1900:
		tonUpperTimeOutFive.IN :=TRUE;
		_fbDiameterMovement.Execute :=TRUE	;	
		IF _fbDiameterMovement.PickDone THEN
			tonUpperTimeOutFive.IN :=FALSE;
			FeedBack.SecondBoxCameraDiameter:=TRUE;
			uiExecutingStep :=2000;
		END_IF
		IF tonUpperTimeOutFive.Q THEN
			_Abort :=TRUE;
			strStatus :='C# DiameterMovement Pickdone timeout';
		END_IF
2000:	//check Second Box CamaraDone
		tonUpperTimeOutFive.IN :=TRUE;
		IF info.SecondBoxCameraDiameterDone THEN
			tonUpperTimeOutFive.IN :=FALSE;
			FeedBack.SecondBoxCameraDiameter:=FALSE;
			_fbDiameterMovement.bContinue:=TRUE;
			uiExecutingStep :=2100;
		END_IF
		IF tonUpperTimeOutFive.Q THEN
			_Abort :=TRUE;
			strStatus :='C# SecondBoxCameraDiameterDone timeout';
		END_IF		
2100:	
		tonUpperTimeOutFive.IN :=TRUE;
		IF _fbDiameterMovement.Done THEN
			tonUpperTimeOutFive.IN :=FALSE;
			_fbDiameterMovement.Execute:=FALSE;
			uiExecutingStep :=2150;
		END_IF
		IF tonUpperTimeOutFive.Q THEN
			_Abort :=TRUE;
			strStatus :='_fbDiameterMovement Done timeout';
		END_IF
2150:
		IF  Input.bUpCV_BoxArrived_Sensor  AND 
			NOT Input.bUpCV_Block1Detect_Sensor  THEN
			uiExecutingStep :=2200;
		END_IF
2200:	// release box 2 from diameter camera pos
		tonUpperTimeOut.IN :=TRUE;
		tonUpperConveyorDelay.PT:=T#100MS;
		tonUpperConveyorDelay.IN := NOT Input.bUpCV_Block1Detect_Sensor ;
		IF tonUpperConveyorDelay.Q THEN	
			tonUpperConveyorDelay.IN := FALSE;
			Cylinder.List.fbUpCV_Block1.M_Extend();
			Cylinder.List.fbUpCV_DiameterPress.M_Retract();		
			Cylinder.List.fbUpCV_Block2.M_Retract();
			uiExecutingStep :=2300;
		END_IF
		IF tonUpperTimeOut.Q THEN
			_Error :=TRUE;
			strStatus := 'There is a box on Input.bUpCV_Block1Detect_Sensor '; 
		END_IF
		
		
2300:
		tonUpperTimeOut.IN :=TRUE;
		IF 	Cylinder.List.fbUpCV_DiameterPress.InRearPosition AND
			Cylinder.List.fbUpCV_Block1.InFrontPosition AND
			Cylinder.List.fbUpCV_Block2.InRearPosition THEN
			tonUpperTimeOut.IN :=FALSE;
			uiExecutingStep :=2500;
		END_IF	
		IF tonUpperTimeOut.Q THEN
			_Error :=TRUE;
			strStatus :='BlockBox1 MoveForward or BlockBox2 MoveBackward or DiameterMeasurementPressBox MoveBackward timeout';
		END_IF
2400:	//Check Box1 in FeedInBox1Detecting and Box2 leave BlockBox2Detecting
		
		tonUpperConveyorDelay.PT:=T#200MS;
		tonUpperConveyorDelay.IN := Input.bUpCV_BoxArrived_Sensor ;
		
		IF  tonUpperConveyorDelay.Q AND NOT Input.bUpCV_Block1Detect_Sensor  THEN
			tonUpperConveyorDelay.IN:=FALSE;
			Cylinder.List.fbUpCV_CamaraPress1.M_Retract();
			Cylinder.List.fbUpCV_Block3.M_Retract();
			Cylinder.List.fbUpCV_Block1.M_Extend();
			uiExecutingStep :=2500;
		END_IF
		
2500:	// Check Box1 in FeedInBox1Sensor and Box2 in BlockBox1Sensor
		tonUpperTimeOutFive.IN :=TRUE;
		tonUpperConveyorDelay.PT:=T#1000MS;
		tonUpperConveyorDelay.IN := Input.bUpCV_BoxArrived_Sensor  AND 
		(Input.bUpCV_Block1Detect_Sensor  OR NOT SecondBox);
		
		IF tonUpperConveyorDelay.Q THEN
			tonUpperTimeOutFive.IN :=FALSE;
			tonUpperConveyorDelay.IN :=FALSE;
			Cylinder.List.fbUpCV_FeedInPress1.M_Extend();
			IF SecondBox THEN
				Cylinder.List.fbUpCV_FeedInPress2.M_Extend();
			END_IF
			uiExecutingStep :=2600;
		END_IF
		IF tonUpperTimeOutFive.Q THEN
			_Error :=TRUE;
			strStatus :='FeedInBox1Detecting not have a box';
		END_IF
2600:
		tonUpperConveyorDelay.PT:=T#500MS;
		tonUpperTimeOut.IN := TRUE;
		tonUpperConveyorDelay.IN :=  Cylinder.List.fbUpCV_FeedInPress1.InFrontPosition AND
		 (Cylinder.List.fbUpCV_FeedInPress2.InFrontPosition OR NOT SecondBox);		
//		IF tonUpperConveyorDelay.IN THEN
//			iMoveConveyor:=0;
//			//Motor.list.UpCV.M_StopMotor();
//		END_IF
		IF tonUpperConveyorDelay.Q THEN
			iMoveConveyor:=0;
			tonUpperTimeOut.IN :=FALSE;
			tonUpperConveyorDelay.IN :=FALSE;
			 Cylinder.List.fbUpCV_FeedInPress1.M_Retract();
			IF SecondBox THEN
				Cylinder.List.fbUpCV_FeedInPress2.M_Retract();
			END_IF
			uiExecutingStep :=2700;
		END_IF	
		IF tonUpperTimeOut.Q THEN
			_Error :=TRUE;
			strStatus :=' Cylinder.List.fbUpCV_FeedInPress1 or Cylinder.List.fbUpCV_FeedInPress2 MoveForward timeout';
		END_IF
2700:
		tonUpperTimeOut.IN :=TRUE;
		IF TON_CheckHaveBox.IN THEN	// conveyor behind not have box feedback 0
			FeedBack.ActualNrOfBox:=0;
		ELSIF SecondBox THEN
			FeedBack.ActualNrOfBox:=2;
			ELSE
			FeedBack.ActualNrOfBox:=1;	
		END_IF
		//Cylinder.List.fbUpCV_Block1.M_Retract();
		//Cylinder.List.fbUpCV_CamaraPress2.M_Retract();
		IF NOT input.bUpCV_ReLoadDetect_Sensor  THEN
			FeedBack.InterventionRequest :=TRUE;
		END_IF
		IF// Cylinder.List.fbUpCV_Block1.InRearPosition AND
			 Cylinder.List.fbUpCV_FeedInPress1.InRearPosition AND
			Cylinder.List.fbUpCV_FeedInPress2.InRearPosition THEN
			//Cylinder.List.fbUpCV_CamaraPress2.InRearPosition THEN
			tonUpperTimeOut.IN :=FALSE;
			uiExecutingStep := 2800;
		END_IF	
		IF tonUpperTimeOut.Q THEN 
			_Error :=TRUE;
			strStatus :='FeedInPressBox1Cylinder or FeedInPressBox2Cylinder or ReadCodePressBox2Cylinder MoveBackward timeout';
		END_IF
		
2800:	//TO check the camera photo speed recoeding time
	TSaveTime 		:= TON_RecordTimer.ET;
	tRecordTimer[iArrayNumber] 			:=TSaveTime;
	tRecordFirstTimer[iArrayNumber] 	:=TSaveFirstTime;
	tRecordSecondTimer[iArrayNumber] 	:=TSaveSecondTime;
	uiExecutingStep := 2900;
2900:
	iArrayNumber := iArrayNumber+1;
	TON_RecordTimer.IN := FALSE;
	IF iArrayNumber >= 101 THEN
		bResetRecordInfo 	:=TRUE;
		iArrayNumber 		:=1;
	END_IF
	uiExecutingStep := 9999;
9999:
	bResetRecordInfo :=FALSE;
	TON_CheckHaveBox.IN :=FALSE;
	_Executed := TRUE;
				
END_CASE
	
	
IF NOT Execute THEN
	eState:=STATE_RESETTING;
END_IF
IF _Error THEN
	//FUN_UniqueErrorCodeGenerator(iErrorID := ErrorID,UinqueErrorCode=>_UniqueErrorCode);
	eState:=STATE_ERROR;
END_IF
IF _Abort OR Abort THEN
	//FUN_UniqueErrorCodeGenerator(iErrorID := ErrorID,UinqueErrorCode=>_UniqueErrorCode);
	eSTATE:=STATE_ABORTING;
END_IF
IF _Executed THEN
	eSTATE:=STATE_Done;
END_IF
END_METHOD

METHOD  M_STATE_RESETTING
VAR_INPUT
END_VAR
Error :=_Error;
Done :=_Executed;

tonUpperTimeOut.IN:=TRUE;
Motor.List.UpCV.M_MotorStop();

IF tonUpperTimeOut.Q OR NOT _Error THEN
	CASE uiResettingStep OF
		0: 
			IF _Error THEN
				Cylinder.List.fbUpCV_Block1.M_Retract();
			END_IF
			Cylinder.List.fbUpCV_FeedInPress1 .M_Retract();	
			Cylinder.List.fbUpCV_FeedInPress2.M_Retract();
			Cylinder.List.fbUpCV_DiameterPress.M_Retract();
			Cylinder.List.fbUpCV_CamaraPress1.M_Retract();	
			//UpperReadCodePressBox2Cylinder.M_Retract();	
			Cylinder.List.fbUpCV_Block2.M_Retract();	
			Cylinder.List.fbUpCV_Block3.M_Retract();	
			Cylinder.List.fbUpCV_CamaraPress4.M_Retract();
			OutPut.bCamara_Blow :=FALSE;
			_fbDiameterMovement.Execute := FALSE;
			_fbDiameterMovement.bContinue:=FALSE;
			FeedBack.InterventionRequest :=FALSE;
			FeedBack.FirstBoxCamera :=FALSE;
			FeedBack.FirstBoxCameraDiameter :=FALSE;
			FeedBack.SecondBoxCamera :=FALSE;
			FeedBack.SecondBoxCameraDiameter :=FALSE;

		
			uiResettingStep:=9999;
		
		9999:
			_ResetCompleted:=TRUE;
	END_CASE
END_IF
IF _ResetCompleted THEN
	eSTATE:=STATE_DORMANT;
END_IF
END_METHOD

END_FUNCTION_BLOCK

// ---- Library/20_MachineUnits/21_StorageArea/Service/FB_AddBoxes_v2.TcPOU
FUNCTION_BLOCK FB_AddBoxes_v2 EXTENDS FB_ObjectBase_V2
VAR_INPUT
//	UpperBoxRefillDetection		:REFERENCE TO FB_Sensor;
//	RackPusherCylinder			:REFERENCE TO FB_Cylinder;
//	RackMotor					:REFERENCE TO FB_RackMotor_V2;
//	bUpperLayerFeedInConveyor	:REFERENCE TO FB_Motor;
	Cylinder 	: REFERENCE TO UNI_CylinderList;
	Motor	 	: REFERENCE TO UNI_MotorList;
	Input 	 	: REFERENCE TO ST_InputTable;
	OutPut	 	: REFERENCE TO ST_OutputTable;
	CurrentData      : ST_SetupPara;

	ERackState	:E_RackState;
	bClearInterventionRequest : BOOL;
	_bForceUpperCV_Use		:BOOL;
END_VAR
VAR_OUTPUT
	InterventionRequest	 : BOOL;
	FeedingBoxes		:BOOL;
END_VAR
VAR
	RackMotorStationTable   : ARRAY[0..9] OF st_StationPositions;
	uiMaxRackStation :INT :=10;
//	eState :E_MethodStatus_Basic;
//	uiExecutingStep : UDINT; // This var is used to been controll STATE_EXECUTING process.
//	uiResettingStep : UDINT;
//	uiAbortingStep : UDINT;
//	_Executed :BOOL; // Executing process completed.
//	_Error : BOOL; // FB has an error.
//	_ResetCompleted : BOOL; // FB resetting completed.
//	_AbortCompleted : BOOL; // FB aborting completed.	

	tonAddBoxTimeOut	:TON;
	tonDetectSensor		:TON;
	tonConveyorTimeOut	:TON;
	tonFeedInUseAddBoxesDelay :TON;
	strStatus	:STRING;
	_Abort		:BOOL;
	uiResumeStep : UINT;
	CurrStation : UINT;
	bInterventionRequest	 : BOOL;
	trigClearInterventionRequest : R_TRIG;
	_bClearInterventionRequestLast :BOOL;
	ftrigRackStateLeaveFeedBox		:F_Trig;	
	_UniqueErrorCode : STRING;
END_VAR

A00_BasicUnits();
SUPER^.A10_StateControl();

ACTION A00_BasicUnits:
tonAddBoxTimeOut(PT:=T#120S);
tonDetectSensor(PT:=T#1S);
tonConveyorTimeOut(PT:=T#5S);
tonFeedInUseAddBoxesDelay(PT:=T#1S);
ErrorID := 2700;

InterventionRequest:=bInterventionRequest;
ftrigRackStateLeaveFeedBox(CLK := (eRackState = E_RackState.FeedBox));
IF ftrigRackStateLeaveFeedBox.Q THEN
	bInterventionRequest:=FALSE;
END_IF

FeedingBoxes := eRackState=E_RackState.FeedBox;
END_ACTION

METHOD PRIVATE M_CheckCommand : BOOL
VAR_INPUT
END_VAR
M_CheckCommand	:= true;
END_METHOD

METHOD PRIVATE M_GetCurrentStation : BOOL
VAR
	i : UINT;
	SetPos	 :LREAL;
END_VAR

VAR_OUTPUT
	uiCurrentStation	:UINT;
END_VAR
//SetPos := THIS^.fbMotor.NcToPlc.SetPos;
SetPos := arAxisCtrl_gb[AxisNo.RackMotor].Admin.Axis.NcToPlc.SetPos;
M_RefreshStationPos();
//IF  THIS^.fbMotor.Status.Homed THEN
IF arAxisCtrl_gb[AxisNo.RackMotor].Admin.Axis.Status.Homed THEN
	FOR i:=0 TO 9 BY 1 DO 
		IF SetPos> RackMotorStationTable[i].Position-5 AND SetPos< RackMotorStationTable[i].Position+5 THEN // Range should be confirm
			uiCurrentStation :=i;
			M_GetCurrentStation :=TRUE;
			RETURN;
		END_IF
	END_FOR
	
	uiCurrentStation:=99;
	M_GetCurrentStation :=FALSE;
ELSE
	M_GetCurrentStation :=FALSE;
	uiCurrentStation:=99;
END_IF
END_METHOD

METHOD PRIVATE M_MoveToStation : BOOL
VAR_INPUT
	uiStation : UINT;
END_VAR
VAR
	bDone	:BOOL;
	uiTargetPosition	:LREAL ;
END_VAR
M_RefreshStationPos();
IF uiStation>=0 AND uiStation <10 THEN
	uiTargetPosition :=RackMotorStationTable[uiStation].Position;
	
	arAxisCtrl_gb[AxisNo.RackMotor].PosMode.Acc := CurrentData.Axes.RackMotor.HalfAuto.Acceleration;
	arAxisCtrl_gb[AxisNo.RackMotor].PosMode.Dec := CurrentData.Axes.RackMotor.HalfAuto.Deceleration;
	arAxisCtrl_gb[AxisNo.RackMotor].PosMode.Jerk := CurrentData.Axes.RackMotor.HalfAuto.Jerk;
	arAxisCtrl_gb[AxisNo.RackMotor].PosMode.Velocity := CurrentData.Axes.RackMotor.HalfAuto.Velocity;
	arAxisCtrl_gb[AxisNo.RackMotor].PosMode.Position := uiTargetPosition;
	
//	THIS^.fbMotor.MoveAbs(lrPosition	:=uiTargetPosition,
//						lrVelocity 		:=GVL.MotorCore[AxisNo.RackMotor].VCC,
//						lrAcceleration	:=GVL.MotorCore[AxisNo.RackMotor].ACC,
//						lrDeceleration	:=GVL.MotorCore[AxisNo.RackMotor].DCC,
//						lrJerk			:=GVL.MotorCore[AxisNo.RackMotor].Jerk,
//						BufferMode		:=MC_BufferMode.MC_Aborting);
	//THIS^.fbMotor.GetCmdDoneStatus(bMotionCmdDone=>bDone);
ELSE
	M_MoveToStation :=FALSE;
	RETURN;
END_IF
END_METHOD

METHOD PRIVATE M_RefreshStationPos : BOOL
VAR_INPUT
END_VAR
VAR
	i: UINT;
	position : ST_PositionTable;
END_VAR
FOR i := 0 TO 9 DO
	position :=FUN_GetPositionTableData(PositionName:='W',Index:=i,Clip:=0);
RackMotorStationTable[i].Position:= position.X_Pos;
END_FOR
	M_RefreshStationPos :=TRUE;

// todo : update position of each stations
//FOR i:=1 TO 200 BY 1 DO
//	FOR iIndex:=0 TO 9 BY 1 DO
//		IF 		
//			DAS_CoreSys.MachineControl.CurrentData.PositionTable[i].Index= iIndex AND
//			DAS_CoreSys.MachineControl.CurrentData.PositionTable[i].Zone ='W' THEN
//			RackMotorStationTable[iIndex].Position := DAS_CoreSys.MachineControl.CurrentData.PositionTable[i].X_Pos;

//			StationsPosition[iIndex]:=RackMotorStationTable[i].Position;
//		ELSE
//			M_RefreshStationPos :=FALSE;
//		END_IF
//	END_FOR
//END_FOR
END_METHOD

METHOD  M_STATE_ABORTED
VAR_INPUT
END_VAR
Error :=TRUE;
Busy :=FALSE;
Done := FALSE;
Status :=strStatus;
UniqueErrorCode:=_UniqueErrorCode;
if not Execute then
	eState := STATE_RESETTING;
END_IF
IF Execute AND Reset THEN
	_Abort := FALSE;
	uiExecutingStep:=uiResumeStep;
	eState:=STATE_EXECUTING;
END_IF
END_METHOD

METHOD  M_STATE_ABORTING
VAR_INPUT
END_VAR
CASE uiAbortingStep of
 0:
 	Cylinder.List.fbStackPush.M_Reset();

	//RackMotor.fbMotor.Reset();	
	
	uiAbortingStep:=9999;
	
9999:	
	_AbortCompleted:=TRUE;
END_CASE

IF	 _AbortCompleted THEN
	eSTATE:=STATE_ABORTED;
END_IF
END_METHOD

METHOD  M_STATE_DONE
VAR_INPUT
END_VAR
Busy := FALSE;
Done := TRUE;
IF NOT Execute THEN
	eState := STATE_RESETTING;
END_IF
END_METHOD

METHOD  M_STATE_DORMANT
VAR_INPUT
END_VAR
VAR
END_VAR
Busy    := FALSE;
Done    := FALSE;
Aborted := FALSE;
Error   := FALSE;
strStatus  := 'No error';
uiExecutingStep := 0;
uiResettingStep := 0;
uiAbortingStep:=0;
uiResumeStep:=0;
_ResetCompleted := FALSE;
_Abort := _Executed := _Error:= _ResetCompleted:=_AbortCompleted:=FALSE;
tonAddBoxTimeOut.IN :=FALSE;
tonDetectSensor.IN:=FALSE;
tonFeedInUseAddBoxesDelay.IN :=FALSE;
_UniqueErrorCode :='0';

IF Execute  THEN 
	IF eRackState = E_RackState.FeedBox THEN
		eState:= STATE_ERROR;
		strStatus :='Rack occupied by user Push FeedButton';
		
	ELSIF  Input.bUpCV_ReLoadDetect_Sensor THEN
		_Executed :=TRUE;
		eState	:= STATE_Done;
	ELSE
		eState := STATE_EXECUTING;
	END_IF	
END_IF
END_METHOD

METHOD  M_STATE_ERROR
VAR_INPUT
END_VAR
Error := TRUE;
Busy :=FALSE;
Status :=strStatus;
UniqueErrorCode:=_UniqueErrorCode;
IF NOT Execute THEN
	eSTATE :=STATE_RESETTING;
END_IF
END_METHOD

METHOD  M_STATE_EXECUTING
VAR_INPUT
END_VAR
VAR_INST
	uiTargetStation	: UINT;
	bMoveConveyor	:BOOL;
END_VAR
VAR
	bMotionDone : BOOL;
	
END_VAR
Busy := TRUE; 
IF NOT _bForceUpperCV_Use THEN
	IF bMoveConveyor THEN
		Motor.List.UpCV.M_MoveForward();	
//	ELSE		
//		Motor.List.UpCV.M_MotorStop();	
	END_IF
END_IF
CASE uiExecutingStep OF			
	0:		//check command
		tonAddBoxTimeOut.IN:=FALSE;
		tonFeedInUseAddBoxesDelay.IN :=TRUE;
			IF M_CheckCommand() THEN
				IF tonFeedInUseAddBoxesDelay.Q THEN
					tonFeedInUseAddBoxesDelay.IN :=FALSE;
					uiExecutingStep	:= 10 ;
				END_IF
			ELSE
				strStatus := 'Wrong command, check the command setting';
				_Error := TRUE;
			END_IF
	10:

		IF 	NOT	Motor.List.UpCV.InBackWard THEN
			uiExecutingStep	:= 100 ;
		END_IF
		//todo : Add timeout
		
 	100:	//release cylinder, check rackmotor currentStation
		tonAddBoxTimeOut.IN:=TRUE;
		tonDetectSensor.IN:=FALSE;
		Cylinder.List.fbStackPush.M_Retract();
		M_GetCurrentStation(uiCurrentStation =>CurrStation);
		
		IF	Cylinder.List.fbStackPush.InRearPosition THEN
		 CASE CurrStation OF
			0 ,99 :
				uiTargetStation:=1;				
			1,2,3,4,5,6,7,8,9 :
				uiTargetStation :=CurrStation;	
			
			ELSE // Error
	
	 	 END_CASE
		END_IF
		
		uiExecutingStep	:= 200 ;
		IF tonAddBoxTimeOut.Q THEN
			strStatus := 'RackPusher move back timeout';
			uiResumeStep:=100;
            _Abort := TRUE;
		END_IF
		
	200:	//check rackmotor station 
		tonDetectSensor.IN :=FALSE;
		IF uiTargetStation<10 THEN
			M_MoveToStation(uiTargetStation);
			uiExecutingStep := 210;	
		ELSE
			uiExecutingStep := 500;	
		END_IF
		
	
	210:
		tonAddBoxTimeOut.IN:=TRUE;
		bMotionDone:= arAxisStatus_gb[AxisNo.RackMotor].Admin._OpModeAck = ModePosAbs AND arAxisStatus_gb[AxisNo.RackMotor].Admin.CmdDone;
	//	RackMotor.fbMotor.GetCmdDoneStatus(bMotionCmdDone=>bMotionDone);
		M_GetCurrentStation(uiCurrentStation =>CurrStation);
	//CurrStation:= RackMotor.P_CurrentStattion;
		IF bMotionDone AND uiTargetStation = CurrStation THEN
			tonAddBoxTimeOut.IN:=FALSE;
			uiExecutingStep := 300;	
		END_IF
		IF tonAddBoxTimeOut.Q THEN
			strStatus := 'Rackmotor moving timeout';
            _Error := TRUE;
		END_IF
		
	300:	//Cylinder moveforward
		tonAddBoxTimeOut.IN:=TRUE;
		Cylinder.List.fbStackPush.M_Extend();
		//bUpperLayerFeedInConveyor.M_ForwardMotor('');
		bMoveConveyor :=TRUE; //Move conveyor motor forward
		IF  Motor.List.UpCV.InForWard THEN	// make sure upperCV release force use
			IF Cylinder.List.fbStackPush.InFrontPosition THEN
				tonAddBoxTimeOut.IN:=FALSE;
				uiExecutingStep := 400;
			END_IF
		END_IF
		IF tonAddBoxTimeOut.Q THEN
			strStatus := 'RackPusher move forward timeout';
			uiResumeStep:=300;
            _Abort := TRUE;
		END_IF
		
	400:	//check refillsensor have refill
		tonDetectSensor.IN:= NOT Input.bUpCV_ReLoadDetect_Sensor;
		Cylinder.List.fbStackPush.M_Retract();
		IF Cylinder.List.fbStackPush.InRearPosition THEN
			IF Input.bUpCV_ReLoadDetect_Sensor THEN
				uiExecutingStep :=500;
			ELSIF tonDetectSensor.Q THEN
				uiTargetStation := CurrStation+1;		
				uiExecutingStep :=200;
			END_IF
		END_IF
		
	500:	//確認氣缸是否在後，Done
		tonAddBoxTimeOut.IN:=TRUE;
			//bUpperLayerFeedInConveyor.M_StopMotor(''); 
			//bMoveConveyor :=FALSE;// Stop Conveyor
			tonAddBoxTimeOut.IN:=FALSE;
			IF uiTargetStation>=9 THEN
				uiExecutingStep :=600;
			ELSE
				bMoveConveyor :=FALSE;
				Motor.List.UpCV.M_MotorStop();	
				uiExecutingStep :=1000;
			END_IF
		
		
		IF tonAddBoxTimeOut.Q THEN
			strStatus := 'RackPusher move back timeout';
			uiResumeStep:=400;
            _Abort := TRUE;
		END_IF
	600:
		tonAddBoxTimeOut.IN:=FALSE	;
		 M_MoveToStation(0);
		 uiExecutingStep:=610;
		 
	610:	
		M_GetCurrentStation(uiCurrentStation =>CurrStation);
		tonAddBoxTimeOut.IN:=TRUE;
		bMotionDone:=arAxisStatus_gb[AxisNo.RackMotor].Admin._OpModeAck = ModePosAbs AND arAxisStatus_gb[AxisNo.RackMotor].Admin.CmdDone;
		IF bMotionDone AND 0 = CurrStation THEN
			bInterventionRequest	 :=TRUE;
			tonAddBoxTimeOut.IN:=FALSE	;
			bMoveConveyor :=FALSE;
			Motor.List.UpCV.M_MotorStop();	
			uiExecutingStep:=1000;
		END_IF
 		IF tonAddBoxTimeOut.Q THEN
			strStatus := 'RackPusher move back timeout';
			uiResumeStep:=400;
            _Abort := TRUE;
		END_IF
	1000:
		bMoveConveyor :=FALSE;// Stop Conveyor
		uiExecutingStep:=1100;
		
	1100:		
		_Executed := TRUE;
	
		
//		strStatus := 'Rack is empty';
//		_Error :=TRUE;
	
	
END_CASE

IF NOT Execute THEN
	eSTATE :=STATE_RESETTING;
END_IF
IF _Executed THEN
	eSTATE := STATE_DONE;
END_IF
IF _Error THEN
	//FUN_UniqueErrorCodeGenerator(iErrorID := ErrorID,UinqueErrorCode=>_UniqueErrorCode);
	eSTATE:=STATE_ERROR;
END_IF
IF _Abort OR Abort THEN
	//FUN_UniqueErrorCodeGenerator(iErrorID := ErrorID,UinqueErrorCode=>_UniqueErrorCode);
	eSTATE:=STATE_ABORTING;
END_IF
END_METHOD

METHOD  M_STATE_RESETTING
VAR_INPUT
END_VAR

VAR
	bMotionDone : BOOL;
END_VAR
CASE uiResettingStep OF
	0:
		tonAddBoxTimeOut.IN:=FALSE;		
		tonDetectSensor.IN:=FALSE;
		Cylinder.List.fbStackPush.M_Retract();

		IF Cylinder.List.fbStackPush.InRearPosition THEN
		uiResettingStep :=100;
		END_IF
		
	100:
		arAxisCtrl_gb[AxisNo.RackMotor].Admin._OpMode.en := E_AXIS_MODE.ModeAH;
		//RackMotor.fbMotor.Stop(0,0);
		//RackMotor.fbMotor.GetCmdDoneStatus(bMotionCmdDone=>bMotionDone);
		Motor.List.UpCV.M_MotorStop();
		uiResettingStep := 200;

		
	200:
		 Error :=false;
		_ResetCompleted := TRUE;
END_CASE

IF _ResetCompleted THEN
	eState := STATE_DORMANT;
END_IF
END_METHOD

END_FUNCTION_BLOCK

// ---- Library/20_MachineUnits/21_StorageArea/Service/FB_BoxSupplyCtrl.TcPOU
FUNCTION_BLOCK FB_BoxSupplyCtrl EXTENDS FB_ObjectBase_V2
VAR_INPUT
//    Execute    :BOOL;   // True : This prog will start.
//    Abort      :BOOL;   // True : This prog will be abort.
//    Reset      :BOOL;   // True : This prog will be reset.
//    ObjectName :STRING; // Set this fb name(About it's action)

//	SupplyBTN 				:REFERENCE TO FB_Button;			//2nd machine
//	RackMotor				:REFERENCE TO FB_RackMotor_V2;
//	BoxesPusherCylinder		:REFERENCE TO FB_Cylinder;


	Cylinder				:REFERENCE TO UNI_CylinderList;
	Input 					:REFERENCE TO ST_InputTable;
	Output					:REFERENCE TO ST_OutputTable;
	StroageRegionMode 		:E_UnitMode;
	bAddsBoxRequest 		: BOOL;
	AddBoxes_Status			:ST_AutoAddsBoxesStatus;
	AddBoxes_Ctrl			:ST_AutoAddsBoxesCommand;
	CurrentData 			: ST_SetupPara;
	
END_VAR

VAR_OUTPUT
	RackState : E_RackState;
	AxisRackMotorBTNHomeRequest	:BOOL;
//    Busy    :BOOL;        // True : This prog is running.
//    Done    :BOOL;        // True : Command has been executed.
//    Aborted :BOOL;        // True : This prog is aborted.
//    Error   :BOOL;        // True : This prog has an error.
//    ErrorID :UINT;       // Output ErrorID
//    Status  :T_MaxString; // Output this prog status by string(255bytes)
END_VAR

VAR
//    eState :E_MethodStatus_Basic;
//	uiExecutingStep : UDINT; // This var is used to been controll STATE_EXECUTING process.
//	uiResettingStep : UDINT;
//	uiAbortingStep : UDINT;
//	_Executed :BOOL; // Executing process completed.
//	_Error : BOOL; // FB has an error.
//	_ResetCompleted : BOOL; // FB resetting completed.
//	_AbortCompleted : BOOL; // FB aborting completed.
	RackMotorStationTable   : ARRAY[0..9] OF st_StationPositions;
	uiMaxRackStation :INT :=10;
	_Abort		: BOOL;
	strStatus	: STRING;
	uiResumeStep : UINT;
	ExcutingStep :E_RackState;
	trigBTN			:R_TRIG;
	trigRequest		:R_TRIG;
	tonBtnCtrl		:ton;
	tonBtnMotorCtrl	:ton;
	tonBlinkTimer :TON;
	tonBlink_Internal :TIME :=T#500MS;

END_VAR

A00_BasicUnits();
SUPER^.A10_StateControl();

ACTION A00_BasicUnits:
tonBtnCtrl(PT:=T#5S);
tonBtnMotorCtrl(PT :=T#30S);
ErrorID := 2800;
END_ACTION

METHOD GetModelState
VAR_OUTPUT
    xDone    :BOOL;
    xBusy    :BOOL;
    xError   :BOOL;
    xAborted :BOOL;
    iErrorID :UDINT;
	UniqueErrorCode : STRING;
END_VAR
xDone    := Done;
xBusy    := Busy;
xError   := Error;
xAborted := Abort;
iErrorID := ErrorID;
END_METHOD

METHOD GetName : STRING
GetName := ObjectName;
END_METHOD

METHOD PRIVATE M_Blink : BOOL
VAR_INPUT
	
END_VAR
tonBlinkTimer(IN :=NOT tonBlinkTimer.Q,
				PT := tonBlink_Internal);
IF tonBlinkTimer.Q THEN
	Output.bStorage_StackPushPbLamp := NOT Output.bStorage_StackPushPbLamp;
END_IF
END_METHOD

METHOD PRIVATE M_GetCurrentStation : BOOL
VAR
	i : UINT;
	SetPos	 :LREAL;
END_VAR

VAR_OUTPUT
	uiCurrentStation	:UINT;
END_VAR
//SetPos := THIS^.fbMotor.NcToPlc.SetPos;
SetPos := arAxisCtrl_gb[AxisNo.RackMotor].Admin.Axis.NcToPlc.SetPos;
M_RefreshStationPos();
//IF  THIS^.fbMotor.Status.Homed THEN
IF arAxisCtrl_gb[AxisNo.RackMotor].Admin.Axis.Status.Homed THEN
	FOR i:=0 TO 9 BY 1 DO 
		IF SetPos> RackMotorStationTable[i].Position-5 AND SetPos< RackMotorStationTable[i].Position+5 THEN // Range should be confirm
			uiCurrentStation :=i;
			M_GetCurrentStation :=TRUE;
			RETURN;
		END_IF
	END_FOR
	
	uiCurrentStation:=99;
	M_GetCurrentStation :=FALSE;
ELSE
	M_GetCurrentStation :=FALSE;
	uiCurrentStation:=99;
END_IF
END_METHOD

METHOD PRIVATE M_MoveToStation : BOOL
VAR_INPUT
	uiStation : UINT;
END_VAR
VAR
	bDone	:BOOL;
	uiTargetPosition	:LREAL ;
END_VAR
M_RefreshStationPos();
IF uiStation>=0 AND uiStation <10 THEN
	uiTargetPosition :=RackMotorStationTable[uiStation].Position;
	
	arAxisCtrl_gb[AxisNo.RackMotor].PosMode.Acc := CurrentData.Axes.RackMotor.HalfAuto.Acceleration;
	arAxisCtrl_gb[AxisNo.RackMotor].PosMode.Dec := CurrentData.Axes.RackMotor.HalfAuto.Deceleration;
	arAxisCtrl_gb[AxisNo.RackMotor].PosMode.Jerk := CurrentData.Axes.RackMotor.HalfAuto.Jerk;
	arAxisCtrl_gb[AxisNo.RackMotor].PosMode.Velocity := CurrentData.Axes.RackMotor.HalfAuto.Velocity;
	arAxisCtrl_gb[AxisNo.RackMotor].PosMode.Position := uiTargetPosition;
	
//	THIS^.fbMotor.MoveAbs(lrPosition	:=uiTargetPosition,
//						lrVelocity 		:=GVL.MotorCore[AxisNo.RackMotor].VCC,
//						lrAcceleration	:=GVL.MotorCore[AxisNo.RackMotor].ACC,
//						lrDeceleration	:=GVL.MotorCore[AxisNo.RackMotor].DCC,
//						lrJerk			:=GVL.MotorCore[AxisNo.RackMotor].Jerk,
//						BufferMode		:=MC_BufferMode.MC_Aborting);
	//THIS^.fbMotor.GetCmdDoneStatus(bMotionCmdDone=>bDone);
ELSE
	M_MoveToStation :=FALSE;
	RETURN;
END_IF
END_METHOD

METHOD PRIVATE M_RefreshStationPos : BOOL
VAR_INPUT
END_VAR
VAR
	i: UINT;
	position : ST_PositionTable;
END_VAR
FOR i := 0 TO 9 DO
	position :=FUN_GetPositionTableData(PositionName:='W',Index:=i,Clip:=0);
RackMotorStationTable[i].Position:= position.X_Pos;
END_FOR
	M_RefreshStationPos :=TRUE;

// todo : update position of each stations
//FOR i:=1 TO 200 BY 1 DO
//	FOR iIndex:=0 TO 9 BY 1 DO
//		IF 		
//			DAS_CoreSys.MachineControl.CurrentData.PositionTable[i].Index= iIndex AND
//			DAS_CoreSys.MachineControl.CurrentData.PositionTable[i].Zone ='W' THEN
//			RackMotorStationTable[iIndex].Position := DAS_CoreSys.MachineControl.CurrentData.PositionTable[i].X_Pos;

//			StationsPosition[iIndex]:=RackMotorStationTable[i].Position;
//		ELSE
//			M_RefreshStationPos :=FALSE;
//		END_IF
//	END_FOR
//END_FOR
END_METHOD

METHOD  M_STATE_ABORTED
VAR_INPUT
END_VAR
ERROR :=TRUE;
Busy    := FALSE;
Aborted := TRUE;
Status := strStatus;

IF NOT Execute THEN
	eSTATE:=STATE_RESETTING;
END_IF

IF Execute AND Reset THEN
	uiExecutingStep :=uiResumeStep;
	eSTATE:=STATE_EXECUTING;
END_IF
END_METHOD

METHOD  M_STATE_ABORTING
VAR_INPUT
END_VAR
CASE uiAbortingStep OF
	0 :
		uiAbortingStep:=9999;
	
	9999:	_AbortCompleted:=TRUE;
END_CASE

IF _AbortCompleted THEN	
	eSTATE :=STATE_ABORTED;
END_IF
END_METHOD

METHOD  M_STATE_DONE
VAR_INPUT
END_VAR
Busy 	:= FALSE;
Done	:=TRUE;

IF NOT Execute THEN
	eSTATE:=STATE_RESETTING;
END_IF
END_METHOD

METHOD  M_STATE_DORMANT
VAR_INPUT
END_VAR
Busy            := FALSE;
Done            := FALSE;
Aborted         := FALSE;
Error           := FALSE;
ErrorID         := 0;
Status          := '';
_ResetCompleted := FALSE;
_Error          := FALSE;
_Executed       := FALSE;
strStatus :='No Error';
uiExecutingStep :=uiResettingStep :=uiResumeStep :=0;

IF Execute THEN
	eSTATE:=STATE_EXECUTING;
END_IF
END_METHOD

METHOD  M_STATE_ERROR
VAR_INPUT
END_VAR
ERROR   :=TRUE;
Busy	:=FALSE;
Status := strStatus;
M_TurnOff();
RackState:= E_RackState.idle; // Useless so far
AxisRackMotorBTNHomeRequest :=false;
IF NOT Execute OR Reset THEN // Execute will always on , therefor Reset is only way to recovery from error	
	eSTATE:=STATE_RESETTING;
END_IF
END_METHOD

METHOD  M_STATE_EXECUTING
VAR_INPUT
END_VAR

VAR_INST
	uiTransitingStep : UINT;
	uiTargetStation :UINT :=0;
	bFreeState	  :BOOL;
END_VAR

VAR
	bMotionDone			:BOOL;
	_uiCurrentStation	:UINT;
END_VAR
Busy :=TRUE;	
//IF SupplyBTN.P_IsBTNRef THEN			//2nd machine 
//	trigBTN(CLK:= (SupplyBTN.P_ButtonState));
//END_IF //Make sure BTN is referenced otherwise exception occur

	trigBTN(CLK:= ( Input.bStorage_StackPushPb));
trigRequest(CLK :=(AddBoxes_Status.InterventionRequest AND bFreeState));

// Force state control
IF AddBoxes_Status.Busy OR AddBoxes_Status.Done  THEN	
	ExcutingStep := E_RackState.AddBoxes;
	
ELSIF StroageRegionMode = E_UnitMode.MANUAL AND
	arAxisCtrl_gb[AxisNo.RackMotor].Admin.Axis.Status.HasJob AND
//	  rackmotor.fbMotor.Status.HasJob AND 
	  NOT (ExcutingStep = E_RackState.FeedBox) THEN	
			ExcutingStep := E_RackState.ManualCtrl;

ELSIF	StroageRegionMode = E_UnitMode.MANUAL AND 
		NOT Cylinder.List.fbStackPush.InRearPosition AND
//		BoxesPusherCylinder.P_IsMoving AND 
		NOT	(ExcutingStep = E_RackState.FeedBox) THEN	
			ExcutingStep := E_RackState.ManualCtrl;

			
END_IF

RackState := ExcutingStep;

CASE ExcutingStep OF
	

	E_RackState.idle:
		;	
	E_RackState.AddBoxes:
		//Service AddBox working
		M_TurnOff();
		bFreeState:=FALSE;
		IF NOT AddBoxes_Ctrl.Execute AND NOT AddBoxes_Status.Error  THEN
        	ExcutingStep := E_RackState.Free;
    	END_IF
		
	E_RackState.ManualCtrl:
	//Stroage area in manual and Rack is moving
		M_TurnOff();
		bFreeState:=FALSE;
		IF NOT arAxisCtrl_gb[AxisNo.RackMotor].Admin.Axis.Status.HasJob AND Cylinder.List.fbStackPush.InRearPosition THEN
            ExcutingStep := E_RackState.Free;
        END_IF
		
	E_RackState.FeedBox:
	// FeedBox mode , 
		M_Blink();
		bFreeState:=FALSE;
		AxisRackMotorBTNHomeRequest :=false;
			IF	trigBTN.Q THEN				
				ExcutingStep :=E_RackState.TransitingFree;	
			END_IF
			
	E_RackState.Free:
	// Rack is free , User is allow to ask to suply box by push the suplyBTN
		M_TurnOn();
		bFreeState:=TRUE;
			 IF trigBTN.Q OR trigRequest.Q THEN
				 uiTransitingStep:=0;
				 ExcutingStep := E_RackState.TransitingFeedBox;
			 END_IF

	E_RackState.TransitingFree:
			 IF NOT AddBoxes_Status.InterventionRequest THEN
				 ExcutingStep :=E_RackState.Free;	
			 END_IF
		
	E_RackState.TransitingFeedBox:
	//Transition step , from Free to FeedBox
		//M_Blink();
		M_TurnOff();
		bFreeState:=FALSE;
		AxisRackMotorBTNHomeRequest :=TRUE;
		// todo : if transition step needs different indication of BTN behavior?
		CASE uiTransitingStep OF
		0:
			tonBtnCtrl.IN	:=FALSE;
			tonBtnMotorCtrl.IN :=FALSE;
			uiTransitingStep:=5;
			M_GetCurrentStation(uiCurrentStation =>_uiCurrentStation);
			IF uiTargetStation = _uiCurrentStation THEN
				uiTransitingStep :=30;
			END_IF
			
		5:	//Move cylinder back
			tonBtnCtrl.IN:=TRUE;			
			Cylinder.List.fbStackPush.M_Retract();
			IF Cylinder.List.fbStackPush.InRearPosition AND NOT arAxisCtrl_gb[AxisNo.RackMotor].Admin.Axis.Status.HasJob THEN 
				tonBtnCtrl.IN :=FALSE;
				uiTransitingStep :=10;
			END_IF
			IF tonBtnCtrl.Q THEN
				_Error:= TRUE;
				StrStatus :='Cylinder MoveBackward timeout';
			END_IF
		10:	// Rackmotor move to station 0
			tonBtnMotorCtrl.IN :=TRUE;
			M_MoveToStation(uiTargetStation);
			IF arAxisCtrl_gb[AxisNo.RackMotor].Admin.Axis.Status.HasJob THEN
				tonBtnMotorCtrl.IN :=FALSE;
			uiTransitingStep :=20;
			END_IF
			IF tonBtnMotorCtrl.Q THEN
				_Error :=TRUE;
				StrStatus :='RackMotor MoveToStation timeout';
			END_IF
		20:	// check currentstation 
			tonBtnMotorCtrl.IN :=TRUE;
//			bMotionDone :=rackmotor.fbMotor.Status.InTargetPosition;
			bMotionDone :=arAxisCtrl_gb[AxisNo.RackMotor].Admin.Axis.Status.InTargetPosition;
			M_GetCurrentStation(uiCurrentStation =>_uiCurrentStation);
			IF bMotionDone  AND uiTargetStation = _uiCurrentStation THEN
				
				uiTransitingStep :=30;
			END_IF
			IF tonBtnMotorCtrl.Q THEN
				_Error :=TRUE;
				StrStatus :='RackMotor currentStation timeout';
			END_IF
		30:
			tonBtnMotorCtrl.IN :=FALSE;
			ExcutingStep := E_RackState.FeedBox;
			AxisRackMotorBTNHomeRequest :=FALSE;
		END_CASE
		


END_CASE
	
IF NOT Execute THEN
	eState:=STATE_RESETTING;
END_IF
IF _Error THEN
	eState:=STATE_ERROR;
END_IF
IF _Abort THEN
	eSTATE:=STATE_ABORTING;
END_IF
IF _Executed THEN
	eSTATE:=STATE_Done;
END_IF
END_METHOD

METHOD  M_STATE_RESETTING
VAR_INPUT
END_VAR
Error :=FALSE;
Done :=FALSE;
Busy := FALSE;
AxisRackMotorBTNHomeRequest :=FALSE;
tonBtnCtrl.IN := FALSE;
tonBtnMotorCtrl.IN := FALSE;
M_TurnOff();
CASE uiResettingStep OF
	
	0:
		uiResettingStep:=9999;


	9999:
		_ResetCompleted:=TRUE;
END_CASE
IF _ResetCompleted THEN
	eSTATE:=STATE_DORMANT;
END_IF
END_METHOD

METHOD PRIVATE M_TurnOff : BOOL
VAR_INPUT
END_VAR
Output.bStorage_StackPushPbLamp := false;
END_METHOD

METHOD PRIVATE M_TurnOn : BOOL
VAR_INPUT
END_VAR
Output.bStorage_StackPushPbLamp := true;
END_METHOD

END_FUNCTION_BLOCK

// ---- Library/20_MachineUnits/23_ShippingArea/FB_ShippingArea.TcPOU
FUNCTION_BLOCK FB_ShippingArea EXTENDS FB_ModeBase_V2 IMPLEMENTS I_UnitState
VAR_INPUT
	FanucRobot : REFERENCE TO FB_FanucRobot_Basic;
	Service : REFERENCE TO ST_ShippingService;
	INPUT       : REFERENCE TO ST_InputTable;
	Motor    : REFERENCE TO UNI_MotorList;
    Reset            : REFERENCE TO BOOL;
	Stop :  REFERENCE TO BOOL;
    bStopMem :  REFERENCE TO BOOL;
END_VAR
VAR_OUTPUT
	Homed : BOOL;
	RobotResetCMD : BOOL;
END_VAR
VAR
	fbShippingRobot_TransmitCVEnd :FB_ShippingRobot_TransmitCVEnd;
	fbShippingRobot_Left : FB_ShippingRobot_Left;
	fbShippingRobot_Right : FB_ShippingRobot_Right;
	fbShippingHoming : FB_ShippingHoming;
END_VAR

SUPER^();

IF __ISVALIDREF(PackTag) THEN
    eModeCommand  := PackTag.Command.UnitMode;
    eStateCommand := PackTag.Command.CntrlCmd;
ELSE
    RETURN;
END_IF

ACTION A00_Service:
fbShippingRobot_TransmitCVEnd(
	Execute:= Service.AutoMode_ShippingRobot_TransmitCVEnd.Command.Execute, 
	Abort:= Service.AutoMode_ShippingRobot_TransmitCVEnd.Command.Abort, 
	Reset:= Reset, 
	ObjectName:= 'Shipping Fanuc Robot TransmitCVEnd', 
	INPUT:=INPUT,
	Motor :=Motor,
	Busy=> Service.AutoMode_ShippingRobot_TransmitCVEnd.Status.Busy, 
	Done=> Service.AutoMode_ShippingRobot_TransmitCVEnd.Status.Done, 
	Aborted=> , 
	Error=> Service.AutoMode_ShippingRobot_TransmitCVEnd.Status.Error, 
	ErrorID=> , 
	Status=> Service.AutoMode_ShippingRobot_TransmitCVEnd.Status.Status, 
	UniqueErrorCode=> , 
	Robot:= FanucRobot, 
	Info:= Service.AutoMode_ShippingRobot_TransmitCVEnd.Info, 
	Stop:= bStopMem);
	
fbShippingRobot_Left(
	Execute:= service.AutoMode_ShippingRobot_Left.Command.Execute, 
	Abort:= Service.AutoMode_ShippingRobot_Left.Command.Abort, 
	Reset:= Reset, 
	ObjectName:= 'Shipping Fanuc Robot Left', 
	Busy=> Service.AutoMode_ShippingRobot_Left.Status.Busy, 
	Done=> Service.AutoMode_ShippingRobot_Left.Status.Done, 
	Aborted=> , 
	Error=> Service.AutoMode_ShippingRobot_Left.Status.Error, 
	ErrorID=> , 
	Status=> Service.AutoMode_ShippingRobot_Left.Status.Status, 
	UniqueErrorCode=> , 
	Robot:= FanucRobot, 
	Info:= Service.AutoMode_ShippingRobot_Left.Info, 
	Stop:=bStopMem);
	
fbShippingRobot_Right(
	Execute:= Service.AutoMode_ShippingRobot_Right.Command.Execute, 
	Abort:= Service.AutoMode_ShippingRobot_Right.Command.Abort, 
	Reset:= Reset, 
	ObjectName:= 'Shipping Fanuc Robot Right', 
	Busy=> Service.AutoMode_ShippingRobot_Right.Status.Busy, 
	Done=> Service.AutoMode_ShippingRobot_Right.Status.Done, 
	Aborted=> , 
	Error=> Service.AutoMode_ShippingRobot_Right.Status.Error, 
	ErrorID=> , 
	Status=> Service.AutoMode_ShippingRobot_Right.Status.Status, 
	UniqueErrorCode=> , 
	Robot:= FanucRobot, 
	Info:= Service.AutoMode_ShippingRobot_Right.Info, 
	Stop:= bStopMem);
	
fbShippingHoming(
	xDone=> , 
	xBusy=> , 
	xError=> , 
	xExecute:= , 
	xAbort:= , 
	FanucRobot:= FanucRobot, 
	Homed:= Homed, 
	xAborted=> , 
	iErrorID=> , 
	ErrorMsg=> , 
	RobotResetCMD=> RobotResetCMD);
END_ACTION

METHOD M_Aborted
M_StateComplete();
END_METHOD

METHOD M_Aborting
M_StateComplete();
END_METHOD

METHOD M_Clearing
M_StateComplete();
END_METHOD

METHOD M_Complete
M_StateComplete();
END_METHOD

METHOD M_Completing
M_StateComplete();
END_METHOD

METHOD M_Execute
CASE eModeCurrent OF
	E_UnitMode.Manual:
		;
	E_UnitMode.Auto:
		;
END_CASE
A00_Service();
//M_StateComplete();
END_METHOD

METHOD M_Held
M_StateComplete();
END_METHOD

METHOD M_Holding
M_StateComplete();
END_METHOD

METHOD M_Idle
M_StateComplete();
END_METHOD

METHOD M_Resetting
M_StateComplete();
END_METHOD

METHOD M_StartHoming
VAR_INPUT
END_VAR
fbShippingHoming.xExecute := TRUE;
END_METHOD

METHOD M_Starting
M_StateComplete();
END_METHOD

METHOD M_StopHoming
VAR_INPUT
END_VAR
fbShippingHoming.xExecute := False;
END_METHOD

METHOD M_Stopped
M_StateComplete();
END_METHOD

METHOD M_Stopping
M_StateComplete();
END_METHOD

METHOD M_Suspended
M_StateComplete();
END_METHOD

METHOD M_Suspending
M_StateComplete();
END_METHOD

METHOD M_Undefined
M_StateComplete();
END_METHOD

METHOD M_Unholding
M_StateComplete();
END_METHOD

METHOD M_Unsuspending
M_StateComplete();
END_METHOD

END_FUNCTION_BLOCK

// ---- Library/20_MachineUnits/23_ShippingArea/Service/FB_ShippingRobot_TransmitCVEnd.TcPOU
FUNCTION_BLOCK FB_ShippingRobot_TransmitCVEnd EXTENDS FB_RobotRegionMove_BufferArea
VAR_INPUT
	INPUT       : REFERENCE TO ST_InputTable;
	Motor    	: REFERENCE TO UNI_MotorList;
END_VAR
VAR_OUTPUT
END_VAR
VAR
	//Area : E_RobotArea := E_RobotArea.TransmitCV_End;
	SensorToBeCheck :BIT;
	ConveyorMotor	: REFERENCE TO FB_Motor ;
	tonBoxArriveDelay 	: TON;
END_VAR

SUPER^.A10_StateControl();
A00_BasicUnits();
Area := E_RobotArea.TransmitCV_End;

ACTION A00_BasicUnits:
tonTimeOut(PT:=T#60S);
tonBoxArriveDelay(PT:=T#1S);

ErrorID:=2250;
END_ACTION

METHOD M_CheckCommand : BOOL // True : Command is useful
VAR_INPUT
END_VAR
VAR
	
END_VAR
// Check command paremeter is correct

THIS^.Get :=TRUE; // For this service , robot only pick box from conveyor
UseA := TRUE; // Only clip A avaliable
UseB := FALSE; // No clipB 	
		
	
	
CASE 	LREAL_TO_INT(Info.A_Position) OF	
	
1: // Pick box from Samesize conveyor
	SensorToBeCheck :=INPUT.bSameSizeCV_BoxNearShippingSensor;
	ConveyorMotor	REF= Motor.List.TransmitSameSideCV;
2: // Pick box from diffSize conveyor
	SensorToBeCheck :=INPUT.bDifferentSizeCV_BoxNearShippingSensor;
	ConveyorMotor	REF= Motor.List.TransmitDifferentSideCV;
ELSE
	strStatus:='Wrong command ,Position A Not allow';
			M_CheckCommand:=FALSE;
			RETURN;	

END_CASE
		
M_CheckCommand:=TRUE;
END_METHOD

METHOD M_CheckUnitsNotBusy : BOOL
VAR_INPUT
END_VAR
M_CheckUnitsNotBusy := true;
END_METHOD

METHOD M_CheckUnitsReady : BOOL
VAR_INPUT
END_VAR
M_CheckUnitsReady := true;
END_METHOD

METHOD PRIVATE M_SensorUpdate : BOOL
VAR_INPUT
END_VAR
CASE 	LREAL_TO_INT(Info.A_Position) OF	
	
1: // Pick box from Samesize conveyor
	SensorToBeCheck :=INPUT.bSameSizeCV_BoxNearShippingSensor;
	
2: // Pick box from diffSize conveyor
	SensorToBeCheck :=INPUT.bDifferentSizeCV_BoxNearShippingSensor;

	
	END_CASE
END_METHOD

METHOD  M_STATE_ABORTED
VAR_INPUT
END_VAR
ERROR :=TRUE;
Busy    := FALSE;
Aborted := TRUE;
Status := strStatus;
UniqueErrorCode:=_UniqueErrorCode;
IF NOT Execute THEN
	eSTATE:=STATE_RESETTING;
END_IF

IF Execute AND Reset THEN
	uiExecutingStep :=uiResumeStep;
	PreviousStrStatus := strStatus;
	PreviousErrorCode := _UniqueErrorCode;
	eSTATE:=STATE_EXECUTING;
END_IF
END_METHOD

METHOD  M_STATE_ABORTING
VAR_INPUT
END_VAR
CASE uiAbortingStep OF
	0 :
		uiAbortingStep:=9999;
		ConveyorMotor.M_MotorStop();
		IF strStatus = PreviousStrStatus THEN
			_UniqueErrorCode :=PreviousErrorCode;
		END_IF
		_Abort :=FALSE;
	9999:	_AbortCompleted:=TRUE;
END_CASE

IF _AbortCompleted THEN	
	eSTATE :=STATE_ABORTED;
END_IF
END_METHOD

METHOD  M_STATE_DONE
VAR_INPUT
END_VAR
Busy := FALSE;
Done := TRUE;
IF NOT Execute THEN
    eState := STATE_RESETTING;
END_IF
END_METHOD

METHOD  M_STATE_DORMANT
VAR_INPUT
END_VAR
// Clear FB output
Busy            := FALSE;
Done            := FALSE;
Aborted         := FALSE;
Error           := FALSE;
ErrorID         := 0;
Status          := '';
_ResetCompleted := FALSE;
_Error          := FALSE;
_Executed       := FALSE;

tonTimeOut.IN:=FALSE;
tonBoxArriveDelay.IN :=FALSE;
strStatus :='No Error';
uiExecutingStep :=uiResettingStep :=uiResumeStep :=0;
PreviousStrStatus			 :='';
PreviousErrorCode			 :='';
_UniqueErrorCode	:='0';

// Wait Execute command
IF Execute THEN
    eState := STATE_EXECUTING;
END_IF
END_METHOD

METHOD  M_STATE_ERROR
VAR_INPUT
END_VAR
ERROR   :=TRUE;
Busy	:=FALSE;
Status := strStatus;
UniqueErrorCode:=_UniqueErrorCode;
ConveyorMotor.M_MotorStop();
IF NOT Execute THEN	
eSTATE:=STATE_RESETTING;
END_IF
END_METHOD

METHOD  M_STATE_EXECUTING
VAR_INPUT
END_VAR
VAR_INST
    ActionMode       : E_ReloadRoundBoxAction;
	BoxReady_1st : BOOL;
	BoxReady_2nd : BOOL;
    CarrierReady_1st : BOOL;
    CarrierReady_2nd : BOOL;
    uiBothStep : UINT;
    uiSingleClampStep : UINT;
	Address_A : INT;
	Address_B : INT;
	bMoveConveyorForward:BOOL;
END_VAR
VAR
	WareHouse: INT;
END_VAR
// Set Busy active edit by johnson
Busy := TRUE;
M_SensorUpdate();

IF THIS^.Stop THEN // Pending the timeout when Stop signal occur
	tonTimeout.IN :=FALSE;
END_IF

IF bMoveConveyorForward THEN
	IF NOT ConveyorMotor.InBackWard THEN
		ConveyorMotor.M_MoveForward();
	END_IF
END_IF
// Service Process
CASE uiExecutingStep OF
	0:
        // Clear variable
		bMoveConveyorForward := FALSE;
        ActionMode       := E_ReloadRoundBoxAction.Undefined;
        CarrierReady_1st := FALSE;
        CarrierReady_2nd := FALSE;
        uiBothStep := 0;
		uiSingleClampStep :=0;
		BoxReady_1st := 0;
		BoxReady_2nd := 0;
		tonTimeOut.IN:=FALSE;
        // Check command
        IF M_CheckCommand() THEN
            uiExecutingStep := 10;
		ELSE
			_Error:=TRUE;
        END_IF
    10:
        // Start process, check units first
        IF M_CheckUnitsReady() THEN
            uiExecutingStep := 20;
        END_IF
    20:
        // CHeck units not busy state
        IF M_CheckUnitsNotBusy() THEN
            uiExecutingStep := 100;
        END_IF
   
		
	100: //Move conveyor 
		bMoveConveyorForward:=TRUE;
		ConveyorMotor.M_MoveForward();			
		uiExecutingStep := 1000;		
	
	1000:   
			// Read   coordinate
 			 Address_A := LREAL_TO_INT(Info.A_Position);
			 Address_B := LREAL_TO_INT(Info.B_Position);
			 
			IF UseA AND NOT UseB THEN
				//Only clampA
				uiExecutingStep := 10000;
//			ELSIF NOT UseA AND UseB THEN
//				//Only ClampB 
//				uiExecutingStep := 20000;
//			ELSIF UseA AND UseB THEN
//				//Both Clamps
//				uiExecutingStep := 30000;		
			END_IF
       
    10000: // Only ClampA 
        IF NOT Robot._DI1.Done THEN            
           		BoxReady_1st:=TRUE;				
			    tonBoxArriveDelay.IN := SensorToBeCheck;      		 
				  // Robot Abs move
           		 Robot.M_StartRobotAbsMove(GetBox:=Get,
											UseClampA:=UseA,
											UseClampB:=UseB,
											Area:=Area,
											ClampA_Address:=Address_A,
											ClampB_Address:=Address_B,
											BoxReady_1:=tonBoxArriveDelay.Q,
											BoxReady_2:=BoxReady_2nd);	  
		
        ELSE
			tonTimeOut.IN:=FALSE;
			tonBoxArriveDelay.IN :=FALSE;
            uiExecutingStep := 10080;
        END_IF
			tonTimeOut.IN:=TRUE;
			IF tonTimeOut.Q=TRUE THEN
				tonTimeOut.IN:=FALSE;			
				strStatus :='wait Box Arrived TransCV time out';
				_Error:=TRUE;
			END_IF	
    10080:
        Robot.M_ResetRobotAbsMove(UseA,UseB); // Clear command and go to place box
		tonTimeOut.IN:=TRUE;
        IF NOT Robot._DI1.Done THEN
			tonTimeOut.IN:=FALSE;
            uiExecutingStep := 90000; 
        END_IF
    	IF tonTimeOut.Q=TRUE THEN
			strStatus :='Reset Robot timeout';
			_Error:=TRUE;
		END_IF	
    
//   20000: // Only ClampB
//        IF NOT Robot._DI1.Done THEN           		
//				BoxReady_2nd:=TRUE;				          		 
//				  // Robot Abs move
//           		 Robot.M_StartRobotAbsMove( GetBox:=Get,
//											UseClampA:=UseA,
//											UseClampB:=UseB,
//											Area:=Area,
//											ClampA_Address:=Address_A,
//											ClampB_Address:=Address_B,
//											BoxReady_1:=BoxReady_1st,
//											BoxReady_2:=BoxReady_2nd);	
//        ELSE
//			tonTimeOut.IN:=FALSE;
//            uiExecutingStep := 20080;
//        END_IF
//		tonTimeOut.IN:=TRUE;
//			IF tonTimeOut.Q=TRUE THEN
//				tonTimeOut.IN:=FALSE;			
//				strStatus :='Reset Robot timeout';
//				_Error:=TRUE;
//			END_IF	
//    20080:
//       Robot.M_ResetRobotAbsMove(UseA,UseB);; // Clear command 

//        IF NOT Robot._DI1.Done THEN
//            uiExecutingStep := 99000; 
//        END_IF
//		tonTimeOut.IN:=TRUE;
//		IF tonTimeOut.Q=TRUE THEN
//			strStatus :='Reset Robot timeout';
//			_Error:=TRUE;
//		END_IF	
//    30000: // Both Clamps
        		
		
//		  CASE uiBothStep OF
//           		0://	
//					BoxReady_1st := FALSE;
//					BoxReady_2nd := FALSE;					
//					uiBothStep:=1000;	
	
//				1000:
//						BoxReady_1st:=TRUE;
//						uiBothStep:=2000;
						
//				2000:
//						IF Robot._DI1.Notification THEN
//							uiBothStep:=3000;
//						END_IF
//				3000:
					
					
//						uiBothStep:=9000;	
					
//				9000:
//						BoxReady_2nd:=TRUE;
//						uiBothStep:=9999;
				
//				9999: //Wait		
//        // wait reset
//        END_CASE

//       	  // Robot Abs move
//           		 Robot.M_StartRobotAbsMove( GetBox:=Get,
//											UseClampA:=UseA,
//											UseClampB:=UseB,
//											Area:=Area,
//											ClampA_Address:=Address_A,
//											ClampB_Address:=Address_B,
//											BoxReady_1:=BoxReady_1st,
//											BoxReady_2:=BoxReady_2nd);	
		
		
//        IF Robot._DI1.Done THEN
//			tonTimeOut.IN:=FALSE;
//            uiExecutingStep := 30080;
//        END_IF
//		IF tonTimeOut.Q=TRUE THEN
//				tonTimeOut.IN:=FALSE;			
//				strStatus :='Reset Robot timeout';
//				_Error:=TRUE;
//			END_IF	
//    30080: // Check robot command is clear
        
//        Robot.M_ResetRobotAbsMove(UseA,UseB);

//        IF NOT Robot._DI1.Done THEN
//			tonTimeOut.IN:=FALSE;
//            uiExecutingStep := 99000; // go to place step
//        END_IF    
//   		tonTimeOut.IN:=TRUE;
//		IF tonTimeOut.Q=TRUE THEN
//			strStatus :='Stop Robot timeout';
//			_Error:=TRUE;
//		END_IF	
   90000:
    bMoveConveyorForward:=FALSE;
   	ConveyorMotor.M_MotorStop();
	IF ConveyorMotor.InStopped THEN
		uiExecutingStep := 99000;
	END_IF
    99000: // process done
                Status    := 'Process completed';
        _Executed := TRUE;
END_CASE

IF _Executed THEN
    eState := STATE_DONE;
ELSIF _Error THEN
	//FUN_UniqueErrorCodeGenerator(iErrorID := ErrorID,UinqueErrorCode=>_UniqueErrorCode);
    eState := STATE_ERROR;
ELSIF NOT Execute THEN
    eState := STATE_RESETTING;
END_IF
IF _Abort OR Abort THEN
	//FUN_UniqueErrorCodeGenerator(iErrorID := ErrorID,UinqueErrorCode=>_UniqueErrorCode);
	eSTATE:=STATE_ABORTING;
END_IF
END_METHOD

METHOD  M_STATE_RESETTING
VAR_INPUT
END_VAR
Error :=FALSE;
Done :=FALSE;
Busy := FALSE;


CASE uiResettingStep OF
	
	0:
		tonTimeOut.IN:=FALSE;
		//Robot.M_ResetAllCommand();
		ConveyorMotor.M_MotorStop();
		Robot.M_ResetRobotAbsMove(TRUE,TRUE);
		
		uiResettingStep:=9999;
	9999:
		_ResetCompleted:=TRUE;
END_CASE
IF _ResetCompleted THEN
	eSTATE:=STATE_DORMANT;
END_IF
END_METHOD

END_FUNCTION_BLOCK

// ---- Library/20_MachineUnits/23_ShippingArea/Service/FB_ShippingRobot_Left.TcPOU
FUNCTION_BLOCK FB_ShippingRobot_Left EXTENDS FB_RobotRegionMove_BufferArea
VAR_INPUT
END_VAR
VAR_OUTPUT
END_VAR
VAR
	//Area : E_RobotArea := E_RobotArea.TransmitCV_End;
END_VAR

SUPER^.A10_StateControl();
A00_BasicUnits();
Area := E_RobotArea.ShippingRobotLeft;

ACTION A00_BasicUnits:
tonTimeOut(PT:=T#60S);
ErrorID:=2250;
END_ACTION

METHOD M_CheckCommand : BOOL // True : Command is useful
VAR_INPUT
END_VAR
VAR
	
END_VAR
// Check command paremeter is correct

THIS^.Get :=Info.Get;
UseA := Info.UseA;
UseB := Info.UseB;
//Buffer area
		
		IF UseA AND ( Info.A_Position<1 OR  Info.A_Position>40) THEN
			strStatus:='Wrong command ,Position A Not allow';
			M_CheckCommand:=FALSE;
			RETURN;			
		END_IF		
	
		IF UseB AND( Info.B_Position<1 OR  Info.B_Position>40 )THEN
			strStatus:='Wrong command ,Position B Not allow';
			M_CheckCommand:=FALSE;
			RETURN;			
		END_IF
		
M_CheckCommand:=TRUE;
END_METHOD

METHOD M_CheckUnitsNotBusy : BOOL
VAR_INPUT
END_VAR
M_CheckUnitsNotBusy := true;
END_METHOD

METHOD M_CheckUnitsReady : BOOL
VAR_INPUT
END_VAR
M_CheckUnitsReady := true;
END_METHOD

METHOD  M_STATE_ABORTED
VAR_INPUT
END_VAR
ERROR :=TRUE;
Busy    := FALSE;
Aborted := TRUE;
Status := strStatus;
UniqueErrorCode:=_UniqueErrorCode;
IF NOT Execute THEN
	eSTATE:=STATE_RESETTING;
END_IF

IF Execute AND Reset THEN
	uiExecutingStep :=uiResumeStep;
	PreviousStrStatus := strStatus;
	PreviousErrorCode := _UniqueErrorCode;
	eSTATE:=STATE_EXECUTING;
END_IF
END_METHOD

METHOD  M_STATE_ABORTING
VAR_INPUT
END_VAR
CASE uiAbortingStep OF
	0 :
		uiAbortingStep:=9999;
		IF strStatus = PreviousStrStatus THEN
			_UniqueErrorCode :=PreviousErrorCode;
		END_IF
		_Abort :=FALSE;
	9999:	_AbortCompleted:=TRUE;
END_CASE

IF _AbortCompleted THEN	
	eSTATE :=STATE_ABORTED;
END_IF
END_METHOD

METHOD  M_STATE_DONE
VAR_INPUT
END_VAR
Busy := FALSE;
Done := TRUE;
IF NOT Execute THEN
    eState := STATE_RESETTING;
END_IF
END_METHOD

METHOD  M_STATE_DORMANT
VAR_INPUT
END_VAR
// Clear FB output
Busy            := FALSE;
Done            := FALSE;
Aborted         := FALSE;
Error           := FALSE;
ErrorID         := 0;
Status          := '';
_ResetCompleted := FALSE;
_Error          := FALSE;
_Executed       := FALSE;

tonTimeOut.IN:=FALSE;
strStatus :='No Error';
uiExecutingStep :=uiResettingStep :=uiResumeStep :=0;
PreviousStrStatus			 :='';
PreviousErrorCode			 :='';
_UniqueErrorCode	:='0';

// Wait Execute command
IF Execute THEN
    eState := STATE_EXECUTING;
END_IF
END_METHOD

METHOD  M_STATE_ERROR
VAR_INPUT
END_VAR
ERROR   :=TRUE;
Busy	:=FALSE;
Status := strStatus;
UniqueErrorCode:=_UniqueErrorCode;
IF NOT Execute THEN	
eSTATE:=STATE_RESETTING;
END_IF
END_METHOD

METHOD  M_STATE_EXECUTING
VAR_INPUT
END_VAR
VAR_INST
    ActionMode       : E_ReloadRoundBoxAction;
	BoxReady_1st : BOOL;
	BoxReady_2nd : BOOL;
    CarrierReady_1st : BOOL;
    CarrierReady_2nd : BOOL;
    uiBothStep : UINT;
    uiSingleClampStep : UINT;
	Address_A : INT;
	Address_B : INT;
END_VAR
VAR
	WareHouse: INT;
END_VAR
// Set Busy active edit by johnson
Busy := TRUE;
IF THIS^.Stop THEN // Pending the timeout when Stop signal occur
	tonTimeout.IN :=FALSE;
END_IF
// Service Process
CASE uiExecutingStep OF
	0:
        // Clear variable
        ActionMode       := E_ReloadRoundBoxAction.Undefined;
        CarrierReady_1st := FALSE;
        CarrierReady_2nd := FALSE;
        uiBothStep := 0;
		uiSingleClampStep :=0;
		BoxReady_1st := 0;
		BoxReady_2nd := 0;
		tonTimeOut.IN:=FALSE;
        // Check command
        IF M_CheckCommand() THEN
            uiExecutingStep := 10;
		ELSE
			_Error:=TRUE;
        END_IF
    10:
        // Start process, check units first
        IF M_CheckUnitsReady() THEN
            uiExecutingStep := 20;
        END_IF
    20:
        // CHeck units not busy state
        IF M_CheckUnitsNotBusy() THEN
            uiExecutingStep := 1000;
        END_IF
   
	1000:   
			// Read   coordinate
 			 Address_A := LREAL_TO_INT(Info.A_Position);
			 Address_B := LREAL_TO_INT(Info.B_Position);
			 
			IF UseA AND NOT UseB THEN
				//Only clampA
				uiExecutingStep := 10000;
			ELSIF NOT UseA AND UseB THEN
				//Only ClampB 
				uiExecutingStep := 20000;
			ELSIF UseA AND UseB THEN
				//Both Clamps
				uiExecutingStep := 30000;		
			END_IF
       
    10000: // Only ClampA 
        IF NOT Robot._DI1.Done THEN            
           		BoxReady_1st:=TRUE;				
			          		 
				  // Robot Abs move
           		 Robot.M_StartRobotAbsMove(GetBox:=Get,
											UseClampA:=UseA,
											UseClampB:=UseB,
											Area:=Area,
											ClampA_Address:=Address_A,
											ClampB_Address:=Address_B,
											BoxReady_1:=BoxReady_1st,
											BoxReady_2:=BoxReady_2nd);	  
		
        ELSE
			tonTimeOut.IN:=FALSE;
            uiExecutingStep := 10080;
        END_IF
			tonTimeOut.IN:=TRUE;
			IF tonTimeOut.Q=TRUE THEN
				tonTimeOut.IN:=FALSE;			
				strStatus :='Reset Robot timeout';
				_Error:=TRUE;
			END_IF	
    10080:
        Robot.M_ResetRobotAbsMove(UseA,UseB); // Clear command and go to place box
		tonTimeOut.IN:=TRUE;
        IF NOT Robot._DI1.Done THEN
			tonTimeOut.IN:=FALSE;
            uiExecutingStep := 99000; 
        END_IF
    	IF tonTimeOut.Q=TRUE THEN
			strStatus :='Reset Robot timeout';
			_Error:=TRUE;
		END_IF	
    
   20000: // Only ClampB
        IF NOT Robot._DI1.Done THEN           		
				BoxReady_2nd:=TRUE;				          		 
				  // Robot Abs move
           		 Robot.M_StartRobotAbsMove( GetBox:=Get,
											UseClampA:=UseA,
											UseClampB:=UseB,
											Area:=Area,
											ClampA_Address:=Address_A,
											ClampB_Address:=Address_B,
											BoxReady_1:=BoxReady_1st,
											BoxReady_2:=BoxReady_2nd);	
        ELSE
			tonTimeOut.IN:=FALSE;
            uiExecutingStep := 20080;
        END_IF
		tonTimeOut.IN:=TRUE;
			IF tonTimeOut.Q=TRUE THEN
				tonTimeOut.IN:=FALSE;			
				strStatus :='Reset Robot timeout';
				_Error:=TRUE;
			END_IF	
    20080:
       Robot.M_ResetRobotAbsMove(UseA,UseB);; // Clear command 

        IF NOT Robot._DI1.Done THEN
            uiExecutingStep := 99000; 
        END_IF
		tonTimeOut.IN:=TRUE;
		IF tonTimeOut.Q=TRUE THEN
			strStatus :='Reset Robot timeout';
			_Error:=TRUE;
		END_IF	
    30000: // Both Clamps
        		
		
		  CASE uiBothStep OF
           		0://	
					BoxReady_1st := FALSE;
					BoxReady_2nd := FALSE;					
					uiBothStep:=1000;	
	
				1000:
						BoxReady_1st:=TRUE;
						uiBothStep:=2000;
						
				2000:
						IF Robot._DI1.Notification THEN
							uiBothStep:=3000;
						END_IF
				3000:
					
					
						uiBothStep:=9000;	
					
				9000:
						BoxReady_2nd:=TRUE;
						uiBothStep:=9999;
				
				9999: //Wait		
        // wait reset
        END_CASE

       	  // Robot Abs move
           		 Robot.M_StartRobotAbsMove( GetBox:=Get,
											UseClampA:=UseA,
											UseClampB:=UseB,
											Area:=Area,
											ClampA_Address:=Address_A,
											ClampB_Address:=Address_B,
											BoxReady_1:=BoxReady_1st,
											BoxReady_2:=BoxReady_2nd);	
		
		
        IF Robot._DI1.Done THEN
			tonTimeOut.IN:=FALSE;
            uiExecutingStep := 30080;
        END_IF
		IF tonTimeOut.Q=TRUE THEN
				tonTimeOut.IN:=FALSE;			
				strStatus :='Reset Robot timeout';
				_Error:=TRUE;
			END_IF	
    30080: // Check robot command is clear
        
        Robot.M_ResetRobotAbsMove(UseA,UseB);

        IF NOT Robot._DI1.Done THEN
			tonTimeOut.IN:=FALSE;
            uiExecutingStep := 99000; // go to place step
        END_IF    
   		tonTimeOut.IN:=TRUE;
		IF tonTimeOut.Q=TRUE THEN
			strStatus :='Stop Robot timeout';
			_Error:=TRUE;
		END_IF	
   
    99000: // process done
                Status    := 'Process completed';
        _Executed := TRUE;
END_CASE

IF _Executed THEN
    eState := STATE_DONE;
ELSIF _Error THEN
	//FUN_UniqueErrorCodeGenerator(iErrorID := ErrorID,UinqueErrorCode=>_UniqueErrorCode);
    eState := STATE_ERROR;
ELSIF NOT Execute THEN
    eState := STATE_RESETTING;
END_IF
IF _Abort OR Abort THEN
	//FUN_UniqueErrorCodeGenerator(iErrorID := ErrorID,UinqueErrorCode=>_UniqueErrorCode);
	eSTATE:=STATE_ABORTING;
END_IF
END_METHOD

METHOD  M_STATE_RESETTING
VAR_INPUT
END_VAR
Error :=FALSE;
Done :=FALSE;
Busy := FALSE;


CASE uiResettingStep OF
	
	0:
		tonTimeOut.IN:=FALSE;
		//Robot.M_ResetAllCommand();
		Robot.M_ResetRobotAbsMove(TRUE,TRUE);
		
		uiResettingStep:=9999;
	9999:
		_ResetCompleted:=TRUE;
END_CASE
IF _ResetCompleted THEN
	eSTATE:=STATE_DORMANT;
END_IF
END_METHOD

END_FUNCTION_BLOCK

// ---- Library/20_MachineUnits/23_ShippingArea/Service/FB_ShippingRobot_Right.TcPOU
FUNCTION_BLOCK FB_ShippingRobot_Right EXTENDS FB_RobotRegionMove_BufferArea
VAR_INPUT
END_VAR
VAR_OUTPUT
END_VAR
VAR
	//Area : E_RobotArea := E_RobotArea.TransmitCV_End;
END_VAR

SUPER^.A10_StateControl();
A00_BasicUnits();
Area := E_RobotArea.ShippingRobotRight;

ACTION A00_BasicUnits:
tonTimeOut(PT:=T#60S);
ErrorID:=2250;
END_ACTION

METHOD M_CheckCommand : BOOL // True : Command is useful
VAR_INPUT
END_VAR
VAR
	
END_VAR
// Check command paremeter is correct

THIS^.Get :=Info.Get;
UseA := Info.UseA;
UseB := Info.UseB;
//Buffer area
		
		IF UseA AND ( Info.A_Position<1 OR  Info.A_Position>40) THEN
			strStatus:='Wrong command ,Position A Not allow';
			M_CheckCommand:=FALSE;
			RETURN;			
		END_IF		
	
		IF UseB AND( Info.B_Position<1 OR  Info.B_Position>40 )THEN
			strStatus:='Wrong command ,Position B Not allow';
			M_CheckCommand:=FALSE;
			RETURN;			
		END_IF
		
M_CheckCommand:=TRUE;
END_METHOD

METHOD M_CheckUnitsNotBusy : BOOL
VAR_INPUT
END_VAR
M_CheckUnitsNotBusy := true;
END_METHOD

METHOD M_CheckUnitsReady : BOOL
VAR_INPUT
END_VAR
M_CheckUnitsReady := true;
END_METHOD

METHOD  M_STATE_ABORTED
VAR_INPUT
END_VAR
ERROR :=TRUE;
Busy    := FALSE;
Aborted := TRUE;
Status := strStatus;
UniqueErrorCode:=_UniqueErrorCode;
IF NOT Execute THEN
	eSTATE:=STATE_RESETTING;
END_IF

IF Execute AND Reset THEN
	uiExecutingStep :=uiResumeStep;
	PreviousStrStatus := strStatus;
	PreviousErrorCode := _UniqueErrorCode;
	eSTATE:=STATE_EXECUTING;
END_IF
END_METHOD

METHOD  M_STATE_ABORTING
VAR_INPUT
END_VAR
CASE uiAbortingStep OF
	0 :
		uiAbortingStep:=9999;
		IF strStatus = PreviousStrStatus THEN
			_UniqueErrorCode :=PreviousErrorCode;
		END_IF
		_Abort :=FALSE;
	9999:	_AbortCompleted:=TRUE;
END_CASE

IF _AbortCompleted THEN	
	eSTATE :=STATE_ABORTED;
END_IF
END_METHOD

METHOD  M_STATE_DONE
VAR_INPUT
END_VAR
Busy := FALSE;
Done := TRUE;
IF NOT Execute THEN
    eState := STATE_RESETTING;
END_IF
END_METHOD

METHOD  M_STATE_DORMANT
VAR_INPUT
END_VAR
// Clear FB output
Busy            := FALSE;
Done            := FALSE;
Aborted         := FALSE;
Error           := FALSE;
ErrorID         := 0;
Status          := '';
_ResetCompleted := FALSE;
_Error          := FALSE;
_Executed       := FALSE;

tonTimeOut.IN:=FALSE;
strStatus :='No Error';
uiExecutingStep :=uiResettingStep :=uiResumeStep :=0;
PreviousStrStatus			 :='';
PreviousErrorCode			 :='';
_UniqueErrorCode	:='0';

// Wait Execute command
IF Execute THEN
    eState := STATE_EXECUTING;
END_IF
END_METHOD

METHOD  M_STATE_ERROR
VAR_INPUT
END_VAR
ERROR   :=TRUE;
Busy	:=FALSE;
Status := strStatus;
UniqueErrorCode:=_UniqueErrorCode;
IF NOT Execute THEN	
eSTATE:=STATE_RESETTING;
END_IF
END_METHOD

METHOD  M_STATE_EXECUTING
VAR_INPUT
END_VAR
VAR_INST
    ActionMode       : E_ReloadRoundBoxAction;
	BoxReady_1st : BOOL;
	BoxReady_2nd : BOOL;
    CarrierReady_1st : BOOL;
    CarrierReady_2nd : BOOL;
    uiBothStep : UINT;
    uiSingleClampStep : UINT;
	Address_A : INT;
	Address_B : INT;
END_VAR
VAR
	WareHouse: INT;
END_VAR
// Set Busy active edit by johnson
Busy := TRUE;
IF THIS^.Stop THEN // Pending the timeout when Stop signal occur
	tonTimeout.IN :=FALSE;
END_IF
// Service Process
CASE uiExecutingStep OF
	0:
        // Clear variable
        ActionMode       := E_ReloadRoundBoxAction.Undefined;
        CarrierReady_1st := FALSE;
        CarrierReady_2nd := FALSE;
        uiBothStep := 0;
		uiSingleClampStep :=0;
		BoxReady_1st := 0;
		BoxReady_2nd := 0;
		tonTimeOut.IN:=FALSE;
        // Check command
        IF M_CheckCommand() THEN
            uiExecutingStep := 10;
		ELSE
			_Error:=TRUE;
        END_IF
    10:
        // Start process, check units first
        IF M_CheckUnitsReady() THEN
            uiExecutingStep := 20;
        END_IF
    20:
        // CHeck units not busy state
        IF M_CheckUnitsNotBusy() THEN
            uiExecutingStep := 1000;
        END_IF
   
	1000:   
			// Read   coordinate
 			 Address_A := LREAL_TO_INT(Info.A_Position);
			 Address_B := LREAL_TO_INT(Info.B_Position);
			 
			IF UseA AND NOT UseB THEN
				//Only clampA
				uiExecutingStep := 10000;
			ELSIF NOT UseA AND UseB THEN
				//Only ClampB 
				uiExecutingStep := 20000;
			ELSIF UseA AND UseB THEN
				//Both Clamps
				uiExecutingStep := 30000;		
			END_IF
       
    10000: // Only ClampA 
        IF NOT Robot._DI1.Done THEN            
           		BoxReady_1st:=TRUE;				
			          		 
				  // Robot Abs move
           		 Robot.M_StartRobotAbsMove(GetBox:=Get,
											UseClampA:=UseA,
											UseClampB:=UseB,
											Area:=Area,
											ClampA_Address:=Address_A,
											ClampB_Address:=Address_B,
											BoxReady_1:=BoxReady_1st,
											BoxReady_2:=BoxReady_2nd);	  
		
        ELSE
			tonTimeOut.IN:=FALSE;
            uiExecutingStep := 10080;
        END_IF
			tonTimeOut.IN:=TRUE;
			IF tonTimeOut.Q=TRUE THEN
				tonTimeOut.IN:=FALSE;			
				strStatus :='Reset Robot timeout';
				_Error:=TRUE;
			END_IF	
    10080:
        Robot.M_ResetRobotAbsMove(UseA,UseB); // Clear command and go to place box
		tonTimeOut.IN:=TRUE;
        IF NOT Robot._DI1.Done THEN
			tonTimeOut.IN:=FALSE;
            uiExecutingStep := 99000; 
        END_IF
    	IF tonTimeOut.Q=TRUE THEN
			strStatus :='Reset Robot timeout';
			_Error:=TRUE;
		END_IF	
    
   20000: // Only ClampB
        IF NOT Robot._DI1.Done THEN           		
				BoxReady_2nd:=TRUE;				          		 
				  // Robot Abs move
           		 Robot.M_StartRobotAbsMove( GetBox:=Get,
											UseClampA:=UseA,
											UseClampB:=UseB,
											Area:=Area,
											ClampA_Address:=Address_A,
											ClampB_Address:=Address_B,
											BoxReady_1:=BoxReady_1st,
											BoxReady_2:=BoxReady_2nd);	
        ELSE
			tonTimeOut.IN:=FALSE;
            uiExecutingStep := 20080;
        END_IF
		tonTimeOut.IN:=TRUE;
			IF tonTimeOut.Q=TRUE THEN
				tonTimeOut.IN:=FALSE;			
				strStatus :='Reset Robot timeout';
				_Error:=TRUE;
			END_IF	
    20080:
       Robot.M_ResetRobotAbsMove(UseA,UseB);; // Clear command 

        IF NOT Robot._DI1.Done THEN
            uiExecutingStep := 99000; 
        END_IF
		tonTimeOut.IN:=TRUE;
		IF tonTimeOut.Q=TRUE THEN
			strStatus :='Reset Robot timeout';
			_Error:=TRUE;
		END_IF	
    30000: // Both Clamps
        		
		
		  CASE uiBothStep OF
           		0://	
					BoxReady_1st := FALSE;
					BoxReady_2nd := FALSE;					
					uiBothStep:=1000;	
	
				1000:
						BoxReady_1st:=TRUE;
						uiBothStep:=2000;
						
				2000:
						IF Robot._DI1.Notification THEN
							uiBothStep:=3000;
						END_IF
				3000:
					
					
						uiBothStep:=9000;	
					
				9000:
						BoxReady_2nd:=TRUE;
						uiBothStep:=9999;
				
				9999: //Wait		
        // wait reset
        END_CASE

       	  // Robot Abs move
           		 Robot.M_StartRobotAbsMove( GetBox:=Get,
											UseClampA:=UseA,
											UseClampB:=UseB,
											Area:=Area,
											ClampA_Address:=Address_A,
											ClampB_Address:=Address_B,
											BoxReady_1:=BoxReady_1st,
											BoxReady_2:=BoxReady_2nd);	
		
		
        IF Robot._DI1.Done THEN
			tonTimeOut.IN:=FALSE;
            uiExecutingStep := 30080;
        END_IF
		IF tonTimeOut.Q=TRUE THEN
				tonTimeOut.IN:=FALSE;			
				strStatus :='Reset Robot timeout';
				_Error:=TRUE;
			END_IF	
    30080: // Check robot command is clear
        
        Robot.M_ResetRobotAbsMove(UseA,UseB);

        IF NOT Robot._DI1.Done THEN
			tonTimeOut.IN:=FALSE;
            uiExecutingStep := 99000; // go to place step
        END_IF    
   		tonTimeOut.IN:=TRUE;
		IF tonTimeOut.Q=TRUE THEN
			strStatus :='Stop Robot timeout';
			_Error:=TRUE;
		END_IF	
   
    99000: // process done
                Status    := 'Process completed';
        _Executed := TRUE;
END_CASE

IF _Executed THEN
    eState := STATE_DONE;
ELSIF _Error THEN
	//FUN_UniqueErrorCodeGenerator(iErrorID := ErrorID,UinqueErrorCode=>_UniqueErrorCode);
    eState := STATE_ERROR;
ELSIF NOT Execute THEN
    eState := STATE_RESETTING;
END_IF
IF _Abort OR Abort THEN
	//FUN_UniqueErrorCodeGenerator(iErrorID := ErrorID,UinqueErrorCode=>_UniqueErrorCode);
	eSTATE:=STATE_ABORTING;
END_IF
END_METHOD

METHOD  M_STATE_RESETTING
VAR_INPUT
END_VAR
Error :=FALSE;
Done :=FALSE;
Busy := FALSE;


CASE uiResettingStep OF
	
	0:
		tonTimeOut.IN:=FALSE;
		//Robot.M_ResetAllCommand();
		Robot.M_ResetRobotAbsMove(TRUE,TRUE);
		
		uiResettingStep:=9999;
	9999:
		_ResetCompleted:=TRUE;
END_CASE
IF _ResetCompleted THEN
	eSTATE:=STATE_DORMANT;
END_IF
END_METHOD

END_FUNCTION_BLOCK

// ---- Library/20_MachineUnits/23_ShippingArea/Service/FB_ShippingHoming.TcPOU
FUNCTION_BLOCK FB_ShippingHoming EXTENDS FB_ActionBasic
VAR_INPUT
	xExecute : BOOL;
	xAbort : BOOL;
    FanucRobot : REFERENCE TO FB_FanucRobot_Basic;
	Homed : REFERENCE TO BOOL;
END_VAR
VAR_OUTPUT
	xAborted : BOOL;
	iErrorID : INT;
	ErrorMsg : STRING;
	RobotResetCMD : BOOL;
END_VAR
VAR
	StateBehaviour 		 : CBML.ETrigA;
	uiShippingHomingStep : UINT;
	FanucRobotCheckTon 	 : TON;
	ResetRobotDelay 	 :TON;
	fbExecuteEdgeDetect  :FB_EdgeDetect;
END_VAR

THIS^.IBehaviourModel := StateBehaviour;
StateBehaviour(xExecute := xExecute,
    xDone => xDone,
    xBusy => xBusy,
    xError => xError,
    xAbort := xAbort OR fbExecuteEdgeDetect.xFallingEdge,
    xAborted => xAborted);

//Error Msg
iErrorID := StateBehaviour._model.iErrorID;
ErrorMsg := M_GetErrorMsg(xErrorID := iErrorID);
FanucRobotCheckTon(PT := T#60S);

//Make sure that C# turns off execute to shut down the service
fbExecuteEdgeDetect(xInput :=xExecute);

ResetRobotDelay(PT:=T#300MS);

METHOD CleanupAction
VAR_INPUT
    xAbortProposed : BOOL;
    iErrorIDProposed: INT;
END_VAR
VAR_OUTPUT
    xComplete : BOOL := TRUE;
    xAbort: BOOL := xAbortProposed;
 	iErrorID : INT := iErrorIDProposed;
END_VAR
RobotResetCMD := FALSE;
FanucRobotCheckTon.IN := FALSE;
uiShippingHomingStep := 0;
END_METHOD

METHOD CyclicAction
VAR_INPUT
    itfTimingController : CBML.ITimingController;
END_VAR
VAR_OUTPUT
    xComplete : BOOL := TRUE;
    iErrorID : INT := 0;
END_VAR
xComplete := FALSE;
CASE uiShippingHomingStep OF
	0:
		FanucRobotCheckTon.IN := TRUE;
		IF FanucRobot.Error THEN
			RobotResetCMD := TRUE;
			ResetRobotDelay.IN:=TRUE;
		ELSE
			uiShippingHomingStep := 500;
		END_IF
		IF ResetRobotDelay.Q THEN
			ResetRobotDelay.IN :=FALSE;
			uiShippingHomingStep := 500;
		END_IF
		
		
	500:
		RobotResetCMD := FALSE;
		FanucRobot.OpMode := E_FanucRobotOpMode.RSR02;
		IF FanucRobot.Error THEN
			RobotResetCMD := TRUE;		
		END_IF
		IF FanucRobot._RSR2_Completed THEN
			uiShippingHomingStep := 600;
		END_IF
	600:
		FanucRobot.OpMode := E_FanucRobotOpMode.RSR01;
		IF FanucRobot._RSR1_Ready THEN
			uiShippingHomingStep := 700;
		END_IF
	700:
		FanucRobotCheckTon.IN := FALSE;
		Homed := TRUE;
		xComplete := TRUE;
END_CASE

IF FanucRobotCheckTon.Q THEN
	iErrorID := 4;
END_IF
END_METHOD

METHOD ExitAction
VAR_INPUT
    xAfterCleanup : BOOL;
    xInCopyCode : BOOL;
END_VAR
END_METHOD

METHOD M_GetErrorMsg : T_MaxString
VAR_INPUT
	xErrorID: INT;
END_VAR

VAR
	
END_VAR
CASE xErrorID OF
    0:
        M_GetErrorMsg := 'No Error';
    1:
        M_GetErrorMsg := 'Action time out';
    2:
        M_GetErrorMsg := 'Cylinder not ready';
    3:
        M_GetErrorMsg := 'Motor not ready';
    4:
		M_GetErrorMsg := 'FanucRobot can not homing';
END_CASE
END_METHOD

METHOD ResetAction
VAR_OUTPUT
    xComplete : BOOL := TRUE;
END_VAR
FanucRobotCheckTon.IN := false;
END_METHOD

METHOD StartAction
VAR_OUTPUT
    xComplete : BOOL := TRUE;
	iErrorID : INT := 0;
END_VAR
Homed := FALSE;
FanucRobotCheckTon.IN := FALSE;
uiShippingHomingStep := 0;
END_METHOD

END_FUNCTION_BLOCK

// ---- Library/99_Utilities/FB_TableMove.TcPOU
FUNCTION_BLOCK FB_TableMove EXTENDS FB_ActionBasic
VAR_INPUT
    xExecute    : BOOL;
    xAbort      : BOOL;
    xReset      : BOOL;
    Index       : INT; // PositionTable array index
    CurrentData : REFERENCE TO ST_SetupPara; // Componets setup parameter
    TimeOut     : LREAL := 30; // Unit : s
END_VAR
VAR_OUTPUT
    xAborted : BOOL;
    iErrorID : INT;
    ErrorMsg : T_MaxString;
END_VAR
VAR
    // State Machine
    StateBehaviour  : CBML.ETrigATo;
    CurrentPosition : ST_PositionTable;
	
	Cylinder : UNI_CylinderList;
	Reset_Rtrig : R_TRIG;
	fbExecuteEdgeDetect :FB_EdgeDetect;
END_VAR

THIS^.IBehaviourModel := StateBehaviour;
StateBehaviour(xExecute := xExecute,
               xAbort := xAbort OR fbExecuteEdgeDetect.xFallingEdge,
               udiTimeOut := LREAL_TO_UDINT( TimeOut*1000000),
               xDone => xDone,
               xBusy => xBusy,
               xError => xError,
               xAborted => xAborted);

//Error Msg
iErrorID := StateBehaviour._model.iErrorID;
ErrorMsg := M_GetErrorMsg(xErrorID := iErrorID);

//Make sure that C# turns off execute to shut down the service
fbExecuteEdgeDetect(xInput :=xExecute);

//Reset
Reset_Rtrig(CLK:= xReset);
IF Reset_Rtrig.Q THEN
	StateBehaviour.ResetModel(xCommit:=xReset);
END_IF

METHOD CleanupAction
VAR_INPUT
    xAbortProposed : BOOL;
    iErrorIDProposed: INT;
END_VAR
VAR_OUTPUT
    xComplete : BOOL := TRUE;
    xAbort: BOOL := xAbortProposed;
 	iErrorID : INT := iErrorIDProposed;
END_VAR
END_METHOD

METHOD CyclicAction
VAR_INPUT
    itfTimingController : CBML.ITimingController;
END_VAR
VAR_OUTPUT
    xComplete : BOOL := TRUE;
    iErrorID : INT := 0;
END_VAR
VAR_INST
	AllowAllocateRobotMove : BOOL;
	AllowOutRobotMove : BOOL;
	AllowRoundBeltMove : BOOL;
	AllowTurnTable :BOOL;
END_VAR
///safe check

xComplete := FALSE;
IF CurrentPosition.Robot = 1  THEN
	arAxisCtrl_gb[AxisNo.OutRobot_X].PosMode.Acc := CurrentData.Axes.OutRobot_X.HalfAuto.Acceleration;
	arAxisCtrl_gb[AxisNo.OutRobot_X].PosMode.Dec := CurrentData.Axes.OutRobot_X.HalfAuto.Deceleration;
	arAxisCtrl_gb[AxisNo.OutRobot_X].PosMode.Jerk := CurrentData.Axes.OutRobot_X.HalfAuto.Jerk;
	arAxisCtrl_gb[AxisNo.OutRobot_X].PosMode.Velocity := CurrentData.Axes.OutRobot_X.HalfAuto.Velocity;
	arAxisCtrl_gb[AxisNo.OutRobot_X].PosMode.Position := CurrentPosition.X_Pos;

	arAxisCtrl_gb[AxisNo.OutRobot_Y].PosMode.Acc := CurrentData.Axes.OutRobot_X.HalfAuto.Acceleration;
	arAxisCtrl_gb[AxisNo.OutRobot_Y].PosMode.Dec := CurrentData.Axes.OutRobot_X.HalfAuto.Deceleration;
	arAxisCtrl_gb[AxisNo.OutRobot_Y].PosMode.Jerk := CurrentData.Axes.OutRobot_X.HalfAuto.Jerk;
	arAxisCtrl_gb[AxisNo.OutRobot_Y].PosMode.Velocity := CurrentData.Axes.OutRobot_X.HalfAuto.Velocity;
	arAxisCtrl_gb[AxisNo.OutRobot_Y].PosMode.Position := CurrentPosition.Y_Pos;
	IF arAxisStatus_gb[AxisNo.OutRobot_X].Admin._OpModeAck = ModePosAbs AND arAxisStatus_gb[AxisNo.OutRobot_X].Admin.CmdDone AND 
		arAxisStatus_gb[AxisNo.OutRobot_Y].Admin._OpModeAck = ModePosAbs AND arAxisStatus_gb[AxisNo.OutRobot_Y].Admin.CmdDone THEN
		xComplete := TRUE;
	END_IF

ELSIF CurrentPosition.Robot = 0  THEN
	arAxisCtrl_gb[AxisNo.Allocate_X].PosMode.Acc := CurrentData.Axes.Allocate_X.HalfAuto.Acceleration;
	arAxisCtrl_gb[AxisNo.Allocate_X].PosMode.Dec := CurrentData.Axes.Allocate_X.HalfAuto.Deceleration;
	arAxisCtrl_gb[AxisNo.Allocate_X].PosMode.Jerk := CurrentData.Axes.Allocate_X.HalfAuto.Jerk;
	arAxisCtrl_gb[AxisNo.Allocate_X].PosMode.Velocity := CurrentData.Axes.Allocate_X.HalfAuto.Velocity;
	arAxisCtrl_gb[AxisNo.Allocate_X].PosMode.Position := CurrentPosition.X_Pos;

	arAxisCtrl_gb[AxisNo.Allocate_Y].PosMode.Acc := CurrentData.Axes.Allocate_Y.HalfAuto.Acceleration;
	arAxisCtrl_gb[AxisNo.Allocate_Y].PosMode.Dec := CurrentData.Axes.Allocate_Y.HalfAuto.Deceleration;
	arAxisCtrl_gb[AxisNo.Allocate_Y].PosMode.Jerk := CurrentData.Axes.Allocate_Y.HalfAuto.Jerk;
	arAxisCtrl_gb[AxisNo.Allocate_Y].PosMode.Velocity := CurrentData.Axes.Allocate_Y.HalfAuto.Velocity;
	arAxisCtrl_gb[AxisNo.Allocate_Y].PosMode.Position := CurrentPosition.Y_Pos;
	IF arAxisStatus_gb[AxisNo.Allocate_X].Admin._OpModeAck = ModePosAbs AND arAxisStatus_gb[AxisNo.Allocate_X].Admin.CmdDone AND 
		arAxisStatus_gb[AxisNo.Allocate_Y].Admin._OpModeAck = ModePosAbs AND arAxisStatus_gb[AxisNo.Allocate_Y].Admin.CmdDone THEN
		xComplete := TRUE;
	END_IF

ELSIF CurrentPosition.Robot = 2  THEN
	arAxisCtrl_gb[AxisNo.RoundBelt].PosMode.Acc := CurrentData.Axes.RoundBelt.HalfAuto.Acceleration;
	arAxisCtrl_gb[AxisNo.RoundBelt].PosMode.Dec := CurrentData.Axes.RoundBelt.HalfAuto.Deceleration;
	arAxisCtrl_gb[AxisNo.RoundBelt].PosMode.Jerk := CurrentData.Axes.RoundBelt.HalfAuto.Jerk;
	arAxisCtrl_gb[AxisNo.RoundBelt].PosMode.Velocity := CurrentData.Axes.RoundBelt.HalfAuto.Velocity;
	arAxisCtrl_gb[AxisNo.RoundBelt].PosMode.Position := CurrentPosition.X_Pos;
	IF arAxisStatus_gb[AxisNo.RoundBelt].Admin._OpModeAck = ModePosAbs AND arAxisStatus_gb[AxisNo.RoundBelt].Admin.CmdDone  THEN
		xComplete := TRUE;
	END_IF

ELSIF CurrentPosition.Robot = 3 THEN
	arAxisCtrl_gb[AxisNo.TurnTable].PosMode.Acc := CurrentData.Axes.TurnTable.HalfAuto.Acceleration;
	arAxisCtrl_gb[AxisNo.TurnTable].PosMode.Dec := CurrentData.Axes.TurnTable.HalfAuto.Deceleration;
	arAxisCtrl_gb[AxisNo.TurnTable].PosMode.Jerk := CurrentData.Axes.TurnTable.HalfAuto.Jerk;
	arAxisCtrl_gb[AxisNo.TurnTable].PosMode.Velocity := CurrentData.Axes.TurnTable.HalfAuto.Velocity;
	arAxisCtrl_gb[AxisNo.TurnTable].PosMode.Position := CurrentPosition.X_Pos;
	IF arAxisStatus_gb[AxisNo.TurnTable].Admin._OpModeAck = ModePosAbs AND arAxisStatus_gb[AxisNo.TurnTable].Admin.CmdDone  THEN
		xComplete := TRUE;
	END_IF

ELSIF CurrentPosition.Robot = 4 THEN
	arAxisCtrl_gb[AxisNo.RackMotor].PosMode.Acc := CurrentData.Axes.RackMotor.HalfAuto.Acceleration;
	arAxisCtrl_gb[AxisNo.RackMotor].PosMode.Dec := CurrentData.Axes.RackMotor.HalfAuto.Deceleration;
	arAxisCtrl_gb[AxisNo.RackMotor].PosMode.Jerk := CurrentData.Axes.RackMotor.HalfAuto.Jerk;
	arAxisCtrl_gb[AxisNo.RackMotor].PosMode.Velocity := CurrentData.Axes.RackMotor.HalfAuto.Velocity;
	arAxisCtrl_gb[AxisNo.RackMotor].PosMode.Position := CurrentPosition.X_Pos;
	IF arAxisStatus_gb[AxisNo.RackMotor].Admin._OpModeAck = ModePosAbs AND arAxisStatus_gb[AxisNo.RackMotor].Admin.CmdDone  THEN
		xComplete := TRUE;
	END_IF

END_IF

IF arAxisCtrl_gb[AxisNo.OutRobot_X].Admin.Axis.Status.Error THEN
	iErrorID := 5; // Axis OutRobot_X has error
END_IF
IF arAxisCtrl_gb[AxisNo.OutRobot_Y].Admin.Axis.Status.Error THEN
	iErrorID := 6; // Axis OutRobotY has error
END_IF
IF arAxisCtrl_gb[AxisNo.Allocate_X].Admin.Axis.Status.Error THEN
	iErrorID := 7; // Axis Allocate_X has error
END_IF
IF arAxisCtrl_gb[AxisNo.Allocate_Y].Admin.Axis.Status.Error THEN
	iErrorID := 8; // Axis Allocate_Y has error
END_IF
IF arAxisCtrl_gb[AxisNo.RoundBelt].Admin.Axis.Status.Error THEN
	iErrorID := 9; // Axis RoundBelt has error
END_IF
IF arAxisCtrl_gb[AxisNo.TurnTable].Admin.Axis.Status.Error THEN
	iErrorID := 10; // Axis TurnTable has error
END_IF
END_METHOD

METHOD ExitAction
VAR_INPUT
    xAfterCleanup : BOOL;
    xInCopyCode : BOOL;
END_VAR
END_METHOD

METHOD M_GetErrorMsg : T_MaxString
VAR_INPUT
	xErrorID: INT;
END_VAR

VAR
	
END_VAR
CASE xErrorID OF
    0:
        M_GetErrorMsg := 'No Error';
    1:
        M_GetErrorMsg := 'Action time out';
    2:
        M_GetErrorMsg := 'Position Data invalid';
    3:
        M_GetErrorMsg := 'Index invalid';
    4:
		M_GetErrorMsg := 'Axis is not ready';
    5:
        M_GetErrorMsg := 'Axis OutRobot X has Error';
    6:
        M_GetErrorMsg := 'Axis OutRobot Y has Error';
	7:
		M_GetErrorMsg := 'Axis Allocate_X has error';
	8:
		M_GetErrorMsg := 'Axis Allocate_Y has error';
	9:
		M_GetErrorMsg := 'Axis RoundBelt has error';
	10:
		M_GetErrorMsg := 'Axis TurnTable has error';
END_CASE
END_METHOD

METHOD ResetAction
VAR_OUTPUT
    xComplete : BOOL := TRUE;
END_VAR
END_METHOD

METHOD StartAction
VAR_OUTPUT
    xComplete : BOOL := TRUE;
	iErrorID : INT := 0;
END_VAR
IF Index >= 1 AND Index <= 200 THEN
CurrentPosition := CurrentData.PositionTable[Index];
ELSE
	iErrorID := 3; // Index invalid
	RETURN;
END_IF
//0 : Allocate , 1: OutRobot, 2: RoundBelt , 3: TurnTable, 4: RackMotor
IF CurrentPosition.Robot = 1  THEN		
	IF arAxisCtrl_gb[AxisNo.OutRobot_X].Admin.Axis.Status.NotMoving AND  
		NOT arAxisCtrl_gb[AxisNo.OutRobot_X].Admin.Axis.Status.Error AND 
		arAxisCtrl_gb[AxisNo.OutRobot_Y].Admin.Axis.Status.NotMoving AND
		NOT arAxisCtrl_gb[AxisNo.OutRobot_Y].Admin.Axis.Status.Error
		THEN
		xComplete := TRUE;
	ELSE
		iErrorID := 4; // Axis not ready
	END_IF
ELSIF CurrentPosition.Robot = 0  THEN
	IF arAxisCtrl_gb[AxisNo.Allocate_X].Admin.Axis.Status.NotMoving AND  
		NOT arAxisCtrl_gb[AxisNo.Allocate_X].Admin.Axis.Status.Error AND 
		arAxisCtrl_gb[AxisNo.Allocate_Y].Admin.Axis.Status.NotMoving AND
		NOT arAxisCtrl_gb[AxisNo.Allocate_Y].Admin.Axis.Status.Error
		THEN
		xComplete := TRUE;
	ELSE
		iErrorID := 4; // Axis not ready
	END_IF
ELSIF CurrentPosition.Robot = 2  THEN
	IF arAxisCtrl_gb[AxisNo.RoundBelt].Admin.Axis.Status.NotMoving AND  
		NOT arAxisCtrl_gb[AxisNo.RoundBelt].Admin.Axis.Status.Error THEN
		xComplete := TRUE;
	ELSE
		iErrorID := 4; // Axis not ready
	END_IF
ELSIF CurrentPosition.Robot = 3  THEN
	IF arAxisCtrl_gb[AxisNo.TurnTable].Admin.Axis.Status.NotMoving AND  
		NOT arAxisCtrl_gb[AxisNo.TurnTable].Admin.Axis.Status.Error THEN 
		xComplete := TRUE;
	ELSE
		iErrorID := 4; // Axis not ready
	END_IF
ELSIF CurrentPosition.Robot = 4  THEN
	IF arAxisCtrl_gb[AxisNo.RackMotor].Admin.Axis.Status.NotMoving AND  
		NOT arAxisCtrl_gb[AxisNo.RackMotor].Admin.Axis.Status.Error THEN 
		xComplete := TRUE;
	ELSE
		iErrorID := 4; // Axis not ready
	END_IF
ELSE
	iErrorID := 2; // Position Data invalid
END_IF
END_METHOD

END_FUNCTION_BLOCK

// ---- Library/10_Machine/12_MachineControl/Service/FB_MachineHoming.TcPOU
FUNCTION_BLOCK FB_MachineHoming EXTENDS FB_ActionBasic
VAR_INPUT
	xExecute : BOOL;
	xAbort : BOOL;
    AllocateHome : REFERENCE TO  FB_AllocateAreaHome;
    StorageHome  :REFERENCE TO FB_StorageHoming;
    ShippingHome :REFERENCE TO FB_ShippingHoming;
	AllocateHomed : REFERENCE TO BOOL;
	StorageHomed : REFERENCE TO BOOL;
	ShippingHomed : REFERENCE TO BOOL;
	Homed : REFERENCE TO BOOL;
    TimeOut     : LREAL := 120; // Unit : s
END_VAR
VAR_OUTPUT
	xAborted : BOOL;
	iErrorID : INT;
	ErrorMsg : STRING;
END_VAR
VAR
	StateBehaviour : CBML.ETrigATo;
	uiMachineHomingStep : UINT;
	fbExecuteEdgeDetect :FB_EdgeDetect;
END_VAR

THIS^.IBehaviourModel := StateBehaviour;
StateBehaviour(xExecute := xExecute,
               xAbort := xAbort OR fbExecuteEdgeDetect.xFallingEdge,
               udiTimeOut := LREAL_TO_UDINT( TimeOut*1000000),
               xDone => xDone,
               xBusy => xBusy,
               xError => xError,
               xAborted => xAborted);
			   
//Make sure that C# turns off execute to shut down the service
fbExecuteEdgeDetect(xInput :=xExecute);

iErrorID := StateBehaviour._model.iErrorID;
ErrorMsg := M_GetErrorMsg(xErrorID := iErrorID);

METHOD CleanupAction
VAR_INPUT
    xAbortProposed : BOOL;
    iErrorIDProposed: INT;
END_VAR
VAR_OUTPUT
    xComplete : BOOL := TRUE;
    xAbort: BOOL := xAbortProposed;
 	iErrorID : INT := iErrorIDProposed;
END_VAR
END_METHOD

METHOD CyclicAction
VAR_INPUT
    itfTimingController : CBML.ITimingController;
END_VAR
VAR_OUTPUT
    xComplete : BOOL := TRUE;
    iErrorID : INT := 0;
END_VAR
xComplete := FALSE;
CASE uiMachineHomingStep OF 
	0:
		IF AllocateHome.Homed AND Storagehome.Homed AND Shippinghome.Homed THEN
			Allocatehome.xExecute := TRUE;
			Storagehome.xExecute := TRUE;
			ShippingHome.xExecute := TRUE;
		END_IF
		IF NOT AllocateHome.Homed THEN
			AllocateHome.xExecute := TRUE;
		END_IF
		IF NOT StorageHome.Homed THEN
			StorageHome.xExecute := TRUE;
		END_IF
		IF NOT ShippingHome.Homed THEN
			ShippingHome.xExecute := TRUE;
		END_IF
		uiMachineHomingStep := 100;
	100:
		IF AllocateHome.Homed AND StorageHome.Homed AND ShippingHome.Homed THEN
			uiMachineHomingStep := 200;
		END_IF
	200:
		Homed := TRUE;
		uiMachineHomingStep := 300;
	300:
		xComplete := TRUE;
		// 
END_CASE
END_METHOD

METHOD ExitAction
VAR_INPUT
    xAfterCleanup : BOOL;
    xInCopyCode : BOOL;
END_VAR
END_METHOD

METHOD M_GetErrorMsg : T_MaxString
VAR_INPUT
	xErrorID: INT;
END_VAR

VAR
	
END_VAR
CASE xErrorID OF
    0:
        M_GetErrorMsg := 'No Error';
    1:
        M_GetErrorMsg := 'Action time out';
    2:
        M_GetErrorMsg := 'Position Data invalid';
    3:
        M_GetErrorMsg := 'Index invalid';
    4:
		M_GetErrorMsg := 'Axis is not ready';
    5:
        M_GetErrorMsg := 'Axis OutRobot X has Error';
    6:
        M_GetErrorMsg := 'Axis OutRobot Y has Error';
	7:
		M_GetErrorMsg := 'Axis Allocate_X has error';
	8:
		M_GetErrorMsg := 'Axis Allocate_Y has error';
	9:
		M_GetErrorMsg := 'Axis RoundBelt has error';
	10:
		M_GetErrorMsg := 'Axis TurnTable has error';
END_CASE
END_METHOD

METHOD ResetAction
VAR_OUTPUT
    xComplete : BOOL := TRUE;
END_VAR
END_METHOD

METHOD StartAction
VAR_OUTPUT
    xComplete : BOOL := TRUE;
	iErrorID : INT := 0;
END_VAR
Homed := FALSE;
uiMachineHomingStep := 0;
END_METHOD

END_FUNCTION_BLOCK

// ---- Library/99_Utilities/FB_CylinderManualCtrl.TcPOU
FUNCTION_BLOCK FB_CylinderManualCtrl
VAR_INPUT
	bTrigger	: BOOL;
	Cylinder	: REFERENCE TO  FB_Cylinder; 
END_VAR
VAR_OUTPUT
END_VAR
VAR
	rTrig	:R_TRIG;
	fTrig	:F_TRIG;
END_VAR

rTrig(CLK:=bTrigger);
fTrig(CLK:=bTrigger);

IF rTrig.Q THEN
	Cylinder.M_Extend();
ELSIF fTrig.Q THEN
	Cylinder.M_Retract();
END_IF

END_FUNCTION_BLOCK

// ---- Library/99_Utilities/FB_MotorManualCtrl.TcPOU
{attribute 'hide_all_locals'}
FUNCTION_BLOCK FB_MotorManualCtrl

VAR_INPUT
	bForward	: BOOL;
	bBackward	: BOOL;
	bStop	: BOOL;
	Motor	: REFERENCE TO  FB_Motor; 
END_VAR
VAR_OUTPUT
END_VAR
VAR
	ForWardrTrig	:R_TRIG;
	ForWardfTrig	:F_TRIG;
	
	BackWardrTrig	:R_TRIG;
	BackWardfTrig	:F_TRIG;
	
	
	
END_VAR

ForWardrTrig(CLK:=bForward);
ForWardfTrig(CLK:=bForward);

BackWardrTrig(CLK:=bBackward);
BackWardfTrig(CLK:=bBackward);


IF ForWardrTrig.Q AND NOT bBackward AND NOT bStop THEN
	Motor.M_MoveForward();	
END_IF

IF BackWardrTrig.q AND NOT bForward AND NOT bStop THEN
	Motor.M_MoveBackward();
END_IF

IF bStop OR ForWardfTrig.Q OR BackWardfTrig.Q THEN
	Motor.M_MotorStop();
END_IF

END_FUNCTION_BLOCK

// ---- Library/99_Utilities/ErrorHandling/FB_ErrorHandler.TcPOU
FUNCTION_BLOCK FB_ErrorHandler EXTENDS FB_ActionBasic
VAR_INPUT
    AlarmList : REFERENCE TO ARRAY[1..Tc3_PackML_V2.MaxAlarms] OF ST_Alarm; // 輸入的錯誤信號矩陣
    HMI_AlarmMonitorList : REFERENCE TO ARRAY[0..999] OF ST_Alarm_Tmax;     // 輸出的錯誤信號矩陣
    AlarmHistory : REFERENCE TO ARRAY[1..Tc3_PackML_V2.MaxHistoryAlarms] OF ST_Alarm;
    MaxRecords : INT := 1000;      // 最大記錄數量
    Reset : BOOL;                  // RESET按鈕
    ResetAllAlarms : BOOL;         // 重置所有錯誤
    EnableLogging : BOOL := TRUE;  // 啟動錯誤紀錄
    ResetDelayTime : TIME := T#3S; // RESET後延遲確認時間
END_VAR
VAR_OUTPUT
    ActiveAlarmCount : INT;    // 活動錯誤數量
    TotalRecords : INT;        // 總記錄數量
    SystemStatus : STRING(50); // 系統狀態
    CurrentSeverityLevel : DINT; // 當前最高嚴重程度 (1-7, 7最嚴重)
	IsResetting : BOOL;       // 正在執行RESET程序
END_VAR
VAR
    // 內部變量
    i : INT;
    j : INT;
	k : INT;
    CurrentTime : DATE_AND_TIME;
    LastTriggerState : ARRAY[1..200] OF BOOL; // 上次Trigger狀態記錄
    RisingEdge : ARRAY[1..200] OF BOOL;       // 上升沿檢測
    FallingEdge : ARRAY[1..200] OF BOOL;      // 下降沿檢測
    RecordIndex : INT := 0;                   // 記錄索引
    HistoryIndex : INT := 1;                  // 歷史記錄索引
    // 邊沿檢測功能塊
    R_TRIG_Array : ARRAY[1..200] OF R_TRIG;
    F_TRIG_Array : ARRAY[1..200] OF F_TRIG;

    // 時間相關
    fbLocalSystemTime : FB_LocalSystemTime := (bEnable := TRUE, dwCycle := 30);
	fbNtTime : GETSYSTEMTIME;
	SystemTimeStruct : TIMESTRUCT;
	_PackMLTime : ARRAY[0..6] OF DINT;
    // 排序用的臨時變數
    TempAlarm : ST_Alarm_Tmax;
    bNeedSort : BOOL;
    TempHistoryAlarm : ST_Alarm; // 歷史記錄排序用
    bNeedHistorySort : BOOL;     // 歷史記錄需要排序
    // 時間比較用的變數
    TimeCompareResult : INT;        // -1:j較舊, 0:相等, 1:j較新
    HistoryTimeCompareResult : INT; // 歷史記錄時間比較結果
    TimeIndex : INT;
	 // 確認機制用的變數
    R_TRIG_Reset : R_TRIG;       // RESET按鈕邊沿檢測
    R_TRIG_Start : R_TRIG;       // START按鈕邊沿檢測
    AllAlarmsCleared : BOOL;     // 所有錯誤都已清除
	// 延遲確認機制
    TON_ResetDelay : TON;        // RESET延遲確認計時器
    ResetInProgress : BOOL;      // RESET程序進行中
    ResetPendingList : ARRAY[0..999] OF BOOL; // 待確認清除的錯誤列表
END_VAR


// 主要執行程序
fbLocalSystemTime();
_PackMLTime := TIMESTRUCT_TO_PackMLTime(fbLocalSystemTime.systemTime);

ActiveAlarmCount := 0;

// RESET按鈕邊沿檢測
R_TRIG_Reset(CLK := Reset);

// RESET延遲確認計時器
TON_ResetDelay(IN := ResetInProgress, PT := ResetDelayTime);
IsResetting := ResetInProgress;

// RESET按鈕延遲確認機制
IF R_TRIG_Reset.Q THEN
    // 啟動RESET程序
    ResetInProgress := TRUE;
    
    // 標記所有當前錯誤為待確認狀態
    FOR i := 0 TO TotalRecords - 1 DO
        ResetPendingList[i] := (HMI_AlarmMonitorList[i].ID <> 0);
    END_FOR;
END_IF;

// RESET延遲時間到達，開始確認錯誤狀態
IF TON_ResetDelay.Q AND ResetInProgress THEN
    ResetInProgress := FALSE;
    
    // 延遲確認：檢查每個標記的錯誤是否真正清除
    FOR i := 0 TO TotalRecords - 1 DO
        IF ResetPendingList[i] AND HMI_AlarmMonitorList[i].ID <> 0 THEN
            // 檢查該錯誤在AlarmList中的對應項目是否已經清除
            FOR j := 1 TO Tc3_PackML_V2.MaxAlarms DO
                IF AlarmList[j].ID = HMI_AlarmMonitorList[i].ID THEN
                    // 找到對應的錯誤源
                    IF NOT AlarmList[j].Trigger THEN
                        // 錯誤已清除，可以移到歷史記錄
                        IF HistoryIndex <= Tc3_PackML_V2.MaxHistoryAlarms THEN
                            // 搬移到AlarmHistory
                            AlarmHistory[HistoryIndex].ID := UDINT_TO_DINT(HMI_AlarmMonitorList[i].ID);
                            AlarmHistory[HistoryIndex].Trigger := FALSE;
                            AlarmHistory[HistoryIndex].Category := HMI_AlarmMonitorList[i].Category;
                            AlarmHistory[HistoryIndex].Value := HMI_AlarmMonitorList[i].Value;
                            AlarmHistory[HistoryIndex].Message := HMI_AlarmMonitorList[i].Message;
                            
                            // 複製發生時間
                            AlarmHistory[HistoryIndex].DateTime := HMI_AlarmMonitorList[i].DateTime;
                            
                            // 記錄清除時間
                            AlarmHistory[HistoryIndex].AckDateTime := _PackMLTime;
                            
                            HistoryIndex := HistoryIndex + 1;
                            IF HistoryIndex > Tc3_PackML_V2.MaxHistoryAlarms THEN
                                HistoryIndex := 1;
                            END_IF;
                        END_IF;
                        
                        // 清空HMI記錄
                        HMI_AlarmMonitorList[i].ID := 0;
                        HMI_AlarmMonitorList[i].Trigger := FALSE;
                        HMI_AlarmMonitorList[i].Category := 0;
                        HMI_AlarmMonitorList[i].Value := 0;
                        HMI_AlarmMonitorList[i].Message := '';
                        HMI_AlarmMonitorList[i].DateTime := DT_TO_PackMLTime(DT#1970-01-01-00:00:00);
                        HMI_AlarmMonitorList[i].ackDateTime := DT_TO_PackMLTime(DT#1970-01-01-00:00:00);
                        
                        bNeedSort := TRUE;
                        bNeedHistorySort := TRUE;
					ELSE
						HMI_AlarmMonitorList[i].Message := AlarmList[j].Message;
                    END_IF;
                    EXIT; // 找到對應項目，跳出內層迴圈
                END_IF;
            END_FOR;
        END_IF;
        // 清除待確認標記
        ResetPendingList[i] := FALSE;
    END_FOR;
END_IF;

// 邊沿檢測和錯誤處理
FOR i := 1 TO Tc3_PackML_V2.MaxAlarms DO
    // 上升沿檢測 - 錯誤發生
    R_TRIG_Array[i](CLK := AlarmList[i].Trigger);
    RisingEdge[i] := R_TRIG_Array[i].Q;
    
    // 下降沿檢測 - 錯誤清除
    F_TRIG_Array[i](CLK := AlarmList[i].Trigger);
    FallingEdge[i] := F_TRIG_Array[i].Q;
    
    // 處理錯誤發生 (上升沿)
    IF RisingEdge[i] AND EnableLogging THEN
        // 檢查是否已存在相同的活動錯誤
        j := -1;  // 初始化為-1，表示未找到
        FOR k := 0 TO TotalRecords - 1 DO
            IF HMI_AlarmMonitorList[k].ID = AlarmList[i].ID AND
                HMI_AlarmMonitorList[k].Trigger THEN
                j := k;  // 找到重複錯誤，記錄位置
                EXIT; // 已存在活動錯誤，跳出
            END_IF;
        END_FOR;
        
        // 如果沒有找到重複的活動錯誤，創建新記錄
        IF j = -1 THEN
            // 尋找空的位置插入新錯誤
            FOR k := 0 TO MaxRecords - 1 DO
                IF HMI_AlarmMonitorList[k].ID = 0 THEN
                    // 找到空位置，插入新錯誤
                    HMI_AlarmMonitorList[k].ID := DINT_TO_UDINT(AlarmList[i].ID);
                    HMI_AlarmMonitorList[k].Trigger := TRUE;
                    HMI_AlarmMonitorList[k].Category := AlarmList[i].Category;
                    HMI_AlarmMonitorList[k].Value := AlarmList[i].Value;
                    HMI_AlarmMonitorList[k].Message := AlarmList[i].Message;
                    
                    // 填入發生時間
                    HMI_AlarmMonitorList[k].DateTime := _PackMLTime;
                    HMI_AlarmMonitorList[k].ackDateTime := DT_TO_PackMLTime(DT#1970-01-01-00:00:00);
                    
                    // 更新記錄統計
                    TotalRecords := TotalRecords + 1;
                    bNeedSort := TRUE;
                    
                    EXIT; // 插入完成，跳出迴圈
                END_IF;
            END_FOR;
        END_IF;
    END_IF;
    
    // 處理錯誤清除 - 修正：移除自動清除邏輯
    // 不再監控下降沿自動清除，只等待RESET按鈕手動清除
    // IF FallingEdge[i] AND EnableLogging THEN
    //     // 此段程式碼已移除，改為只在RESET時處理
    // END_IF;
    
    // 統計活動錯誤數量
    IF AlarmList[i].Trigger THEN
        ActiveAlarmCount := ActiveAlarmCount + 1;
    END_IF;
END_FOR;

// 如果有資料異動，重新排序HMI_AlarmMonitorList
// 保持錯誤記錄不被清除，只排序顯示順序
IF bNeedSort THEN
    // 簡化排序：只按時間排序，不清除任何記錄
    FOR i := 0 TO MaxRecords - 2 DO
        FOR j := 0 TO MaxRecords - 2 - i DO
            // 只有兩個位置都有有效記錄才比較
            IF HMI_AlarmMonitorList[j].ID <> 0 AND HMI_AlarmMonitorList[j+1].ID <> 0 THEN
                
                // 比較發生時間，較新的排在前面
                TimeCompareResult := 0;
                FOR TimeIndex := 0 TO 5 DO
                    IF HMI_AlarmMonitorList[j].DateTime[TimeIndex] < HMI_AlarmMonitorList[j+1].DateTime[TimeIndex] THEN
                        TimeCompareResult := -1; // j較舊
                        EXIT;
                    ELSIF HMI_AlarmMonitorList[j].DateTime[TimeIndex] > HMI_AlarmMonitorList[j+1].DateTime[TimeIndex] THEN
                        TimeCompareResult := 1; // j較新
                        EXIT;
                    END_IF;
                END_FOR;
                
                // 如果j較舊，交換位置（較新的往前）
                IF TimeCompareResult = -1 THEN
                    TempAlarm := HMI_AlarmMonitorList[j];
                    HMI_AlarmMonitorList[j] := HMI_AlarmMonitorList[j+1];
                    HMI_AlarmMonitorList[j+1] := TempAlarm;
                END_IF;
            END_IF;
        END_FOR;
    END_FOR;
    
    // 重新計算TotalRecords（所有有效記錄，不管Trigger狀態）
    TotalRecords := 0;
    FOR i := 0 TO MaxRecords - 1 DO
        IF HMI_AlarmMonitorList[i].ID <> 0 THEN
            TotalRecords := TotalRecords + 1;
        END_IF;
    END_FOR;
    
    bNeedSort := FALSE;
END_IF;

// 如果歷史記錄有新資料，重新排序AlarmHistory (使用PackMLTime比較)
IF bNeedHistorySort THEN
    // 使用泡沫排序法排序歷史記錄 (按DateTime由新到舊)
    FOR i := 1 TO Tc3_PackML_V2.MaxHistoryAlarms - 1 DO
        FOR j := 1 TO Tc3_PackML_V2.MaxHistoryAlarms - i DO
            // 只排序有效的記錄 (ID不為0)
            IF AlarmHistory[j].ID <> 0 AND AlarmHistory[j+1].ID <> 0 THEN
                
                // 比較兩個時間：j vs j+1
                HistoryTimeCompareResult := 0;
                
                // 比較PackMLTime陣列
                FOR TimeIndex := 0 TO 5 DO
                    IF AlarmHistory[j].DateTime[TimeIndex] < AlarmHistory[j+1].DateTime[TimeIndex] THEN
                        HistoryTimeCompareResult := -1; // j較舊
                        EXIT;
                    ELSIF AlarmHistory[j].DateTime[TimeIndex] > AlarmHistory[j+1].DateTime[TimeIndex] THEN
                        HistoryTimeCompareResult := 1; // j較新
                        EXIT;
                    END_IF;
                END_FOR;
                
                // 如果j較舊，則交換位置（讓較新的往前移）
                IF HistoryTimeCompareResult = -1 THEN
                    TempHistoryAlarm := AlarmHistory[j];
                    AlarmHistory[j] := AlarmHistory[j+1];
                    AlarmHistory[j+1] := TempHistoryAlarm;
                END_IF;
            END_IF;
        END_FOR;
    END_FOR;
    
    bNeedHistorySort := FALSE;
END_IF;

// 更新系統狀態和嚴重程度
CurrentSeverityLevel := 0; // 初始化為無錯誤

// 掃描HMI_AlarmMonitorList中活動錯誤的最高嚴重程度
FOR i := 0 TO TotalRecords - 1 DO
    IF HMI_AlarmMonitorList[i].Trigger THEN  // 只計算活動錯誤
        // 找出最高嚴重程度
        IF HMI_AlarmMonitorList[i].Value > CurrentSeverityLevel THEN
            CurrentSeverityLevel := HMI_AlarmMonitorList[i].Value;
        END_IF;
    END_IF;
END_FOR;

// 統計真正的活動錯誤數量（Trigger=TRUE）
ActiveAlarmCount := 0;
FOR i := 0 TO TotalRecords - 1 DO
    IF HMI_AlarmMonitorList[i].Trigger THEN
        ActiveAlarmCount := ActiveAlarmCount + 1;
    END_IF;
END_FOR;

END_FUNCTION_BLOCK

// ---- Library/99_Utilities/FB_SignalTower.TcPOU
FUNCTION_BLOCK FB_SignalTower
VAR_INPUT
    // TRUE: Activates the defined operation
    // FALSE: Aborts/resets the defined operation
    Enable     :BOOL := TRUE;
    LampRed    :REFERENCE TO BOOL;
    LampYellow :REFERENCE TO BOOL;
    LampGreen  :REFERENCE TO BOOL;
    Buzz       :REFERENCE TO BOOL;
	ForceCloseBuzz : BOOL;
	BuzzSwitchOnTime	:LREAL :=3000.0 ; //In Second
END_VAR

VAR_OUTPUT
    // TRUE: Operation is running
    Vaild :BOOL;
    // TRUE: Error condition reached
    Error :BOOL;
    // Error code describing error condition
    ErrorID :DINT;
END_VAR

VAR
    LampRed_Active    :BOOL;         // True :Lamp Red actived
    LampYellow_Active :BOOL;         // True :Lamp Yellow actived
    LampGreen_Active  :BOOL;         // True : Lamp Green actived
    FB_1Hz            :FB_SignalGen; // 1Hz flash signal generator
    FB_2Hz            :FB_SignalGen; // 2Hz flash signal generator
    FB_05Hz           :FB_SignalGen; // 0.5 Hz flash signal generator
    // Signal Tower controller output
    LampSingal :ST_SignalTower;
	BuzzOnTimer			:TON;

END_VAR

// Call Signal generator
A_SignalGenerator();

// 
IF Enable THEN
	LampSingal.Lamp_Red 	:= M_LampRed();
	LampSingal.Lamp_Yellow	:= M_LampYellow();
	LampSingal.Lamp_Green 	:= M_LampGreen();
	LampSingal.Buzz			:=M_Buzz(BuzzSwitchOnTime);
ELSE
	LampSingal.Lamp_Red := FALSE;
	LampSingal.Lamp_Yellow := FALSE;
	LampSingal.Lamp_Green := FALSE;
	LampSingal.Buzz := FALSE;
END_IF

LampRed := LampSingal.Lamp_Red;
LampYellow := LampSingal.Lamp_Yellow;
LampGreen := LampSingal.Lamp_Green;
Buzz := LampSingal.Buzz;

ACTION A_SignalGenerator:
FB_1Hz(PT := F_FtoPT(Hz := 1));
FB_2Hz(PT := F_FtoPT(Hz := 2));
FB_05Hz(PT := F_FtoPT(Hz := 0.5));
END_ACTION

METHOD M_Buzz : BOOL
VAR_INPUT
	SwitchOnTime : LREAL ;//In second
END_VAR
VAR
	SignalMode: E_SignalTowerLampMode:=E_SignalTowerLampMode.Disable;
	
END_VAR
BuzzOnTimer(PT:= DWORD_TO_TIME(LREAL_TO_DWORD(SwitchOnTime*1000)));

IF ForceCloseBuzz THEN
	SignalMode := E_SignalTowerLampMode.Disable;
ELSE
	IF  GVL_ADS.MachineState = E_MachineState.Error THEN
		BuzzOnTimer.IN :=TRUE;		
		SignalMode := E_SignalTowerLampMode.Flash_2Hz;			
	ELSE   
		BuzzOnTimer.IN :=FALSE;
	END_IF
	
END_IF
// Determine the Lamp mode based on the current SignalTowerMode. 
CASE SignalMode OF
    E_SignalTowerLampMode.Disable: // Lamp off
        M_Buzz := FALSE;
    E_SignalTowerLampMode.AlwaysOn: // Lamp on
        M_Buzz := TRUE AND NOT BuzzOnTimer.Q;
    E_SignalTowerLampMode.Flash_05Hz: // Lamp flash 0.25s on 0.25s off
        M_Buzz := FB_05Hz.Q AND NOT BuzzOnTimer.Q;
    E_SignalTowerLampMode.Flash_1Hz: // Lamp flash 0.5s on 0.5s off	
        M_Buzz := FB_1Hz.Q AND NOT BuzzOnTimer.Q ;
    E_SignalTowerLampMode.Flash_2Hz: // Lamp flash 1s on 1s off
        M_Buzz := FB_2Hz.Q AND ( NOT BuzzOnTimer.Q);
END_CASE
END_METHOD

METHOD M_LampGreen : BOOL
VAR_INPUT
END_VAR
VAR
	SignalMode: E_SignalTowerLampMode:=E_SignalTowerLampMode.Disable;
END_VAR
IF NOT LampRed_Active  THEN
    IF GVL_ADS.MachineState=E_MachineState.Running THEN
        SignalMode := E_SignalTowerLampMode.AlwaysOn;
    ELSE
        SignalMode := E_SignalTowerLampMode.Disable;
    END_IF
ELSIF LampRed_Active  THEN
    SignalMode := E_SignalTowerLampMode.Disable;
END_IF;

// Determine the Lamp mode based on the current SignalTowerMode. 
CASE SignalMode OF
    E_SignalTowerLampMode.Disable: // Lamp off
        M_LampGreen := FALSE;
    E_SignalTowerLampMode.AlwaysOn: // Lamp on
        M_LampGreen := TRUE;
    E_SignalTowerLampMode.Flash_05Hz: // Lamp flash 0.25s on 0.25s off
        M_LampGreen := FB_05Hz.Q;
    E_SignalTowerLampMode.Flash_1Hz: // Lamp flash 0.5s on 0.5s off	
        M_LampGreen := FB_1Hz.Q;
    E_SignalTowerLampMode.Flash_2Hz: // Lamp flash 1s on 1s off
        M_LampGreen := FB_2Hz.Q;
END_CASE

// Lamp effective flag
IF SignalMode = E_SignalTowerLampMode.Disable THEN
    LampGreen_Active := FALSE;
ELSE
    LampGreen_Active := TRUE;
END_IF
END_METHOD

METHOD M_LampRed : BOOL
VAR_INPUT
END_VAR
VAR
	SignalMode: E_SignalTowerLampMode:=E_SignalTowerLampMode.Disable;
END_VAR
// Control SignalMode here
IF GVL_ADS.MachineState=E_MachineState.Error THEN
	SignalMode := E_SignalTowerLampMode.Flash_1Hz;
ELSIF GVL_ADS.MachineState=E_MachineState.StandBy THEN
	SignalMode := E_SignalTowerLampMode.AlwaysOn;	
ELSE
	SignalMode := E_SignalTowerLampMode.Disable;
END_IF
// Determine the Lamp mode based on the current SignalTowerMode. 
CASE SignalMode OF
    E_SignalTowerLampMode.Disable: // Lamp off
        M_LampRed := FALSE;
    E_SignalTowerLampMode.AlwaysOn:// Lamp on
        M_LampRed := TRUE;
    E_SignalTowerLampMode.Flash_05Hz:// Lamp flash 0.25s on 0.25s off
        M_LampRed := FB_05Hz.Q;
    E_SignalTowerLampMode.Flash_1Hz: // Lamp flash 0.5s on 0.5s off
        M_LampRed := FB_1Hz.Q;
    E_SignalTowerLampMode.Flash_2Hz: // Lamp flash 1s on 1s off
        M_LampRed := FB_2Hz.Q;
END_CASE
// Lamp effective flag
IF SignalMode = E_SignalTowerLampMode.Disable THEN
	LampRed_Active := FALSE;
ELSE
	LampRed_Active := TRUE;
END_IF
END_METHOD

METHOD M_LampYellow : BOOL
VAR_INPUT
END_VAR
VAR
	SignalMode: E_SignalTowerLampMode:=E_SignalTowerLampMode.Disable;
END_VAR
// Contorl Signal here
 IF GVL_ADS.MachineState=E_MachineState.NotHomed OR GVL_ADS.MachineState=E_MachineState.Homing THEN
	
		SignalMode := E_SignalTowerLampMode.Flash_2Hz;
	ELSIF GVL_ADS.MachineState=E_MachineState.Homed THEN
		SignalMode := E_SignalTowerLampMode.AlwaysOn;
	ELSE	
		SignalMode := E_SignalTowerLampMode.Disable;
	
END_IF

// Determine the Lamp mode based on the current SignalTowerMode. 
CASE SignalMode OF
    E_SignalTowerLampMode.Disable: // Lamp off
        M_LampYellow := FALSE;
    E_SignalTowerLampMode.AlwaysOn:// Lamp on
        M_LampYellow := TRUE;
    E_SignalTowerLampMode.Flash_05Hz:// Lamp flash 0.25s on 0.25s off
        M_LampYellow := FB_05Hz.Q;
    E_SignalTowerLampMode.Flash_1Hz: // Lamp flash 0.5s on 0.5s off
        M_LampYellow := FB_1Hz.Q;
    E_SignalTowerLampMode.Flash_2Hz: // Lamp flash 1s on 1s off
        M_LampYellow := FB_2Hz.Q;
END_CASE
// Lamp effective flag
IF SignalMode = E_SignalTowerLampMode.Disable THEN
	LampYellow_Active := FALSE;
ELSE
	LampYellow_Active := TRUE;
END_IF
END_METHOD

PROPERTY PUBLIC P_LampGreenState : Bool
GET
P_LampGreenState:=LampSingal.Lamp_Green ;
END_GET
END_PROPERTY

PROPERTY PUBLIC P_LampRedState : Bool
GET
P_LampRedState:=LampSingal.Lamp_Red ;
END_GET
END_PROPERTY

PROPERTY PUBLIC P_LampYellowState : Bool
GET
P_LampYellowState:=LampSingal.Lamp_Yellow ;
END_GET
END_PROPERTY

END_FUNCTION_BLOCK

// ---- Library/99_Utilities/FB_SignalGen.TcPOU
// This function block allocates 50% of the time to ON and 50% of the time to OFF based on the input time. 
// For example, if the input is 1 second, it generates a signal of 0.5 seconds ON, followed by 0.5 seconds OFF.
FUNCTION_BLOCK FB_SignalGen
VAR_INPUT
	PT : TIME;
END_VAR

VAR_OUTPUT
	Q : BOOL;
END_VAR

VAR
	tn : DWORD;
	tx : DWORD;
	init : BOOL;
END_VAR

tx := TIME_TO_DWORD(TIME());
IF NOT init THEN
	init := TRUE;
	tn := tx;
	Q := TRUE;
ELSIF tx - tn >= SHR(TIME_TO_DWORD(PT), 1) THEN
	Q := NOT Q;
	tn := tn + SHR(TIME_TO_DWORD(pt), 1);
END_IF;

END_FUNCTION_BLOCK

// ---- Library/99_Utilities/F_FtoPT.TcPOU
// Frequence to time(PT is Timer target value)
FUNCTION F_FtoPT : Time
VAR_INPUT
	Hz : REAL;
END_VAR
VAR
END_VAR

IF Hz > 0 THEN
	F_FtoPT := DWORD_TO_TIME(REAL_TO_DWORD((1000 / Hz)));
ELSE
	F_FtoPT := T#0S;
END_IF

END_FUNCTION

// ---- Library/99_Utilities/FUNCTION/FUN_MachineState.TcPOU
FUNCTION FUN_MachineState : E_MachineState
VAR_INPUT
	Error :BOOL;
	Estop : BOOL;
	Stop :BOOL;
	Reset:BOOL;
	Start :BOOL;
	HomeBusy :BOOL;
	Homed :BOOL;
	MachineMode : E_UnitMode;
	eMachineState : E_MachineState;
END_VAR
VAR
		
END_VAR

IF Error OR EStop THEN
	eMachineState:=E_MachineState.Error;
END_IF

CASE eMachineState OF
	E_MachineState.Default :
		eMachineState:=E_MachineState.NotHomed;
	E_MachineState.NotHomed:

		IF HomeBusy THEN
			eMachineState:=E_MachineState.Homing;
		ELSIF Homed THEN
			eMachineState:=E_MachineState.Homed;
		END_IF
	
	E_MachineState.Homing:
		
		IF Homed THEN
			eMachineState:=E_MachineState.Homed;
		END_IF
	
	E_MachineState.Homed:
	
		IF MachineMode = E_UnitMode.AUTO THEN
			eMachineState:=E_MachineState.Running;
		END_IF
		IF HomeBusy THEN
			eMachineState:=E_MachineState.Homing;
		END_IF
		
	E_MachineState.Running:
	
		IF Stop THEN
			eMachineState:=E_MachineState.StandBy;
		END_IF
		
		 IF MachineMode = E_UnitMode.MANUAL THEN
			eMachineState:=E_MachineState.Homed;			
		 END_IF
		 
	E_MachineState.StandBy:
		
		IF Start THEN
			eMachineState:=E_MachineState.Running;
		END_IF
		IF MachineMode = E_UnitMode.MANUAL THEN
			eMachineState:=E_MachineState.Homed;			
		 END_IF
		 
	E_MachineState.Error:
		
		IF Reset OR NOT Error THEN
			eMachineState:=E_MachineState.StandBy;
		END_IF

END_CASE

FUN_MachineState := eMachineState ;

END_FUNCTION

// ---- POUs/DAS_MotionSync.TcPOU
PROGRAM DAS_MotionSync
VAR
END_VAR

AxisInterface_Type03();
M_InputMapping();

